		//DCタイムをゲット
		aPostprocessingDcTime[0]:=F_GetActualDcTime64();
	
		//1 コンテナ初期化
		hr := F_VN_CreateContainer(ipBoundingBoxes, ContainerType_Vector_TcVnRectangle_DINT, cNumBox, hr);		//NMS関数座標用
        hr := F_VN_CreateContainer(ipScores, ContainerType_Vector_REAL, cNumBox, hr);							//NMS関数スコア用
		
		hr := FW_SafeRelease(ADR(GVL.ipResultPoints));															//GVLにあるXY座標入力用コンテナをリリース(初回はコンテナ無いけど、大丈夫な関数)
		hr := F_VN_CreateContainer(GVL.ipResultPoints, ContainerType_Vector_TcVnPoint2_DINT, 0, hr);			//GVLにあるXY座標入力用コンテナ作成

		
		//2 Row Dataを座標用コンテナに書き込み
		nIteratorIdx:=0;		//インデックスリセット
		hr := F_VN_GetForwardIterator(ipBoundingBoxes, ipIterator, hr);		//座標用コンテナから前方走査イテレータを取得
		IF SUCCEEDED(hr) AND ipIterator <> 0 THEN
			hr := ipIterator.TcQueryInterface(IID_ITcVnAccess_TcVnRectangle_DINT, ADR(ipAccessTcVnRectangleDINT));		//TcVnRectangle_DINT型アクセス用のアクセスインターフェースをクエリ
			IF SUCCEEDED(hr) AND ipAccessTcVnRectangleDINT <> 0 THEN
				WHILE SUCCEEDED(hr) AND ipIterator.CheckIfEnd() <> S_OK DO		//コンテナの終端に達するまで高速ループ
					
					stRectangle.nX			:=REAL_TO_DINT(stModelOutput.out_output[0, nIteratorIdx, 0]-(stModelOutput.out_output[0, nIteratorIdx, 2]/2.0));		// 計算式： 左上X ＝ 中心X － (幅 ÷ 2)
					stRectangle.nY			:=REAL_TO_DINT(stModelOutput.out_output[0, nIteratorIdx, 1]-(stModelOutput.out_output[0, nIteratorIdx, 3]/2.0));		// 計算式： 左上Y ＝ 中心Y － (高さ ÷ 2)
					stRectangle.nWidth		:=REAL_TO_DINT(stModelOutput.out_output[0, nIteratorIdx, 2]);
					stRectangle.nHeight		:=REAL_TO_DINT(stModelOutput.out_output[0, nIteratorIdx, 3]);		//YOLOXセンター座標（cx, cy）から、TwinCAT左上座標（x, y）に変換して中間バッファのストラクトに書き込み
				
					hr := ipAccessTcVnRectangleDINT.Set(stRectangle);		//アクセスインターフェース経由でデータをコンテナに書き込み
					
					IF SUCCEEDED(hr) THEN
						hr := ipIterator.Increment();
						nIteratorIdx:=nIteratorIdx+1;
					END_IF
					
				END_WHILE
			END_IF
			hr := FW_SafeRelease(ADR(ipAccessTcVnRectangleDINT));		//アクセスインターフェースを解放
		END_IF 
		hr := FW_SafeRelease(ADR(ipIterator));		//イテレータを解放


		//3 Row Dataをスコア用コンテナに書き込み
		nIteratorIdx:=0;		//インデックスリセット
		hr := F_VN_GetForwardIterator(ipScores, ipIterator, hr);		//スコア用コンテナから前方走査イテレータを取得
		IF SUCCEEDED(hr) AND ipIterator <> 0 THEN
			hr := ipIterator.TcQueryInterface(IID_ITcVnAccess_REAL, ADR(ipAccessREAL));		//REAL型アクセス用のアクセスインターフェースをクエリ
			IF SUCCEEDED(hr) AND ipAccessREAL <> 0 THEN
				WHILE SUCCEEDED(hr) AND ipIterator.CheckIfEnd() <> S_OK DO		//コンテナの終端に達するまで高速ループ
					
					hr := ipAccessREAL.Set(stModelOutput.out_output[0, nIteratorIdx, 4] * stModelOutput.out_output[0, nIteratorIdx, 5]);		//アクセスインターフェース経由でデータをコンテナに書き込み
																																				//スコアはobj_score（物体らしさスコア）× class_score（クラススコア）					
					IF SUCCEEDED(hr) THEN
						hr := ipIterator.Increment();
						nIteratorIdx:=nIteratorIdx+1;
					END_IF
					
				END_WHILE
			END_IF
			hr := FW_SafeRelease(ADR(ipAccessREAL));		//アクセスインターフェースを解放
		END_IF 
		hr := FW_SafeRelease(ADR(ipIterator));		//イテレータを解放
		

		//4 Non-Maximum Suppression (NMS) の実行
        hr := F_VN_NonMaxSuppression(ipBoundingBoxes, ipScores, ipDestIndices, 0.3, 0.45, hr);		// 第4引数 (0.3)、第5引数（0.45）の説明コードの末尾にあり

		//NMS生存結果の抽出・描画・GVL出力
		hr := F_VN_GetNumberOfElements(ipDestIndices, nElementsFound, hr);		//NMSで生き残った（＝検出確定した）ワークの総数をカウント
		
		//1個以上ワークが検出された場合のみ、ループで1個ずつ処理を回す
		IF SUCCEEDED(hr) AND nElementsFound > 0 THEN
			
			FOR nIdx := 0 TO (ULINT_TO_UDINT(nElementsFound) - 1) DO
							
				hr := F_VN_GetAt_DINT(ipDestIndices, nTargetIndex, UDINT_TO_ULINT(nIdx), hr);		//NMSコンテナから、生き残った「元のRowDataのインデックス番号」を抽出

				hr := F_VN_GetAt_TcVnRectangle_DINT(ipBoundingBoxes, stFinalRect, DINT_TO_ULINT(nTargetIndex), hr);		//抽出したインデックスを使って、元の座標コンテナから長方形（Rect）データを取得
				
				hr := F_VN_GetAt_REAL(ipScores, fFinalScore, DINT_TO_ULINT(nTargetIndex), hr);		//抽出したインデックスを使って、元のスコアコンテナから確率データを取得

				// ONNXの座標から余白を引いて、縮小倍率で割り戻すことで、元画像のピクセル位置に戻す
				stFinalRect.nX      :=REAL_TO_DINT((DINT_TO_REAL(stFinalRect.nX) - fPadX) / fScale);
				stFinalRect.nY      :=REAL_TO_DINT((DINT_TO_REAL(stFinalRect.nY) - fPadY) / fScale);
				stFinalRect.nWidth  :=REAL_TO_DINT(DINT_TO_REAL(stFinalRect.nWidth) / fScale);
				stFinalRect.nHeight :=REAL_TO_DINT(DINT_TO_REAL(stFinalRect.nHeight) / fScale);
				
				//ワークの中心座標 (cx, cy) を計算し、DINT型構造体に落とし込む
				stCenterPoint[0]:=stFinalRect.nX + (stFinalRect.nWidth / 2);
				stCenterPoint[1]:=stFinalRect.nY + (stFinalRect.nHeight / 2);
				
				//確率表示にしたいので100倍
				fFinalScore:=fFinalScore*100.0;
				
				//ワーク幅から外れた物は無視
				IF (cWorkWidthMin<stFinalRect.nWidth AND stFinalRect.nWidth<cWorkWidthMax) AND (cWorkWidthMin<stFinalRect.nHeight AND stFinalRect.nHeight<cWorkWidthMax)  THEN
					
					//5 出力画像にワークの位置を画像に書き込み
					hr := F_VN_DrawRectangle(stFinalRect.nX, stFinalRect.nY, stFinalRect.nX+stFinalRect.nWidth, stFinalRect.nY + stFinalRect.nHeight,ipImageOut, aGreen, 2, hr);		//ワークを囲む長方形を描画
					
					hr := F_VN_DrawPoint(stCenterPoint[0], stCenterPoint[1], ipImageOut, TCVN_DS_PLUS, aGreen, hr);		//中心点に十字マークを描画
	
	
					//6 ワークのxy座標を画像に書き込み
					fbFormatString(	sFormat	:='( %2.1f ) = (%.3d, %.3d)', 
									arg1	:=F_REAL(fFinalScore),
									arg2	:=F_DINT(stCenterPoint[0]),
									arg3	:=F_DINT(stCenterPoint[1]));		//書き込み文字列生成
					
					hr := F_VN_PutText(fbFormatString.sOut, ipImageOut, stFinalRect.nX, stFinalRect.nY, TCVN_FT_HERSHEY_TRIPLEX, 0.5, aGreen, hr);		//XY座標を描画
					
					//7 GVLにあるコンテナにxy座標を書き込み
					hr := F_VN_AppendToContainer_TcVnVector2_DINT(stCenterPoint, GVL.ipResultPoints, hr);
				
				END_IF
				
			END_FOR
		END_IF
		
		//DCタイムをゲット
		aPostprocessingDcTime[1]:=F_GetActualDcTime64();
		
		iStep:=11;
		
	6..10:
		//NA

	11:
		//画面表示イメージを作成する
		hr := F_VN_TransformIntoDisplayableImage(ipImageIn, ipImageInDisp, hr);
        hr := F_VN_TransformIntoDisplayableImage(ipImageOut, ipImageOutDisp, hr);

		//ポインターの開放
		FW_SafeRelease(ADR(ipTensorImage));
		FW_SafeRelease(ADR(ipBoundingBoxes));
		FW_SafeRelease(ADR(ipScores));
		FW_SafeRelease(ADR(ipDestIndices));
		
		//各実行時間を計算[ms]
		lrPreprocessingTime		:=ULINT_TO_LREAL(aPreprocessingDcTime[1]-aPreprocessingDcTime[0]) / 1000000.0;
		lrInferenceTime			:=ULINT_TO_LREAL(aInferenceDcTime[1]-aInferenceDcTime[0]) / 1000000.0;
		lrPostprocessingTime	:=ULINT_TO_LREAL(aPostprocessingDcTime[1]-aPostprocessingDcTime[0]) / 1000000.0;
		
        iStep := 0;
		
	END_CASE







(*ワンポイントメモ

NMS処理の引数説明
0.3 ＝ スコアの閾値（足切りライン）正式な引数名はfScoreThreshold
意味：
*直前で計算した「obj_score × class_score」の最終スコアが、「0.3（30%）未満のゴミ候補は、重なりを調べる前に最初から全部切り捨てる」という設定です。
現場での調整イメージ：
*誤検出（ワークがないのに背景を誤認識する）が多いとき			:この値を 0.4 や 0.5 に上げます。より自信のある候補しか残らなくなります。
*見落とし（あるはずのワークをスルーしてしまう）が多いとき		:この値を 0.2 や 0.15 に下げます。少し自信がなくても候補として拾うようになります。

2. 0.45 ＝ 重複の閾値（ダブり判定の基準）正式な引数名は fOverlapThreshold
意味：
*1つのワークに対して、AIが何個もダブって四角枠（ボックス）を出してしまったときに、「面積の45%以上が重なっていたら、それは同じワークを二重検出しているとみなして、スコアが低い方を消す」という設定です。
※この重なりの割合をAIの世界では「IoU（Intersection over Union）」と呼びます。
現場での調整イメージ：
*1つのワークに四角枠が2個も3個も重なって残ってしまうとき								:この値を 0.3 や 0.35 に下げます（重なりの判定を厳しくして、ちょっとでも重なっていたら容赦なく1個にまとめます）。
*ワーク同士が実際に近くに密集していて、隣のワークの枠まで巻き添えで消されてしまうとき	:この値を 0.55 や 0.6 に上げます（かなりガッツリ重なっていない限り、別々のワークとして認めるようになります）。

*)

END_PROGRAM

// ---- 01_Submodules/Axis/FB_AxisVelocity.TcPOU
FUNCTION_BLOCK FB_AxisVelocity
VAR_OUTPUT
	// =============== State variables ========================
	bError			: BOOL;					// Error signal
	nErrorID		: UDINT;				// Error ID
	bMoves			: BOOL;					// Status of moving
END_VAR
VAR	
	// =============== Done signals of Halt and Reset =========
	bResetDone		: BOOL;					// Status of function block MC_Reset
	bHaltDone		: BOOL;					// Status of function block MC_Halt

	// =============== State variables ========================
	bStatusEnable	: BOOL;					// Enable feedback
	
	// =============== Velocity, override =====================
	fVelocity		: LREAL;				// Target velocity
	fOverride 		: LREAL := 100.0;		// Override 100%
	
	// =============== Trigger function blocks ================
	fbTriggerHalt	: R_TRIG;				// Trigger to recognize rising edge of halt input
	fbTriggerReset	: R_TRIG;				// Trigger to recognize rising edge of reset input
	
	// =============== Axis reference =========================
	AxisRef			: AXIS_REF;				// Axis reference (process data plc/nc)
	
	// =============== Motion function blocks =================
	fbMcPower 		: MC_Power;				// FB for enable and override
	fbMcReset 		: MC_Reset;				// FB to reset axis
	fbMcStop 		: MC_Stop;				// FB to stop axis
	fbMcHalt		: MC_Halt;				// FB to halt axis
	fbMcMove		: MC_MoveVelocity;		// FB to move axis (velocity movement)
END_VAR

// =========================================================
;
// =========================================================

PROPERTY bState_Enable : BOOL
GET
bState_Enable := bStatusEnable;
END_GET
END_PROPERTY

PROPERTY bState_HaltDone : BOOL
GET
bState_HaltDone := bHaltDone;
END_GET
END_PROPERTY

PROPERTY bState_ResetDone : BOOL
GET
bState_ResetDone := bResetDone;
END_GET
END_PROPERTY

METHOD Enable
VAR_INPUT
	bEnable		: BOOL;
END_VAR
// =========================================================

fbMCPower(	Enable 			:= bEnable, 
			Enable_Positive	:= bEnable, 
			Enable_Negative	:= bEnable, 
			Override		:= fOverride,
			Axis			:= AxisRef,
			Status			=> bStatusEnable);
			
IF fbMcPower.Error THEN
	bError		:= TRUE;
	nErrorID 	:= fbMcPower.ErrorID;
END_IF

AxisRef.ReadStatus();

bMoves := AxisRef.Status.Moving;

// =========================================================
END_METHOD

PROPERTY fTargetVelocity : LREAL
GET
fTargetVelocity := fVelocity;
END_GET
SET
fVelocity := fTargetVelocity;
END_SET
END_PROPERTY

METHOD Halt
VAR_INPUT
	bDriveHalt		: BOOL;					// Request stop
END_VAR
// =========================================================

IF bDriveHalt THEN
	// Move Execute FALSE
	fbMCMove(	Execute	:= FALSE,
				Axis 	:= AxisRef);
ELSE
	// Reset done signal
	bHaltDone := FALSE;
END_IF

// Trigger
fbTriggerHalt(CLK := bDriveHalt);

IF fbTriggerHalt.Q THEN
	fbMcHalt(	Execute	:= TRUE,
				Axis 	:= AxisRef);
ELSE
	fbMcHalt(Axis := AxisRef);
END_IF

// Done / Error / Command aborted
IF fbMcHalt.Done OR fbMcHalt.Error OR fbMcHalt.CommandAborted THEN
	bError		:= fbMcHalt.Error;
	nErrorID 	:= fbMcHalt.ErrorID;
	bHaltDone 	:= fbMcHalt.Done;
	
	fbMCMove(	Execute	:= FALSE,
				Axis 	:= AxisRef);
				
	fbMcHalt(	Execute	:= FALSE,
				Axis 	:= AxisRef);
END_IF

// =========================================================
END_METHOD

METHOD MoveBw
VAR_INPUT
END_VAR
// =========================================================

// Not error
IF NOT fbMcMove.Error THEN
	fbMCMove(	Execute 	:= TRUE,
				Velocity 	:= fVelocity,
				Direction 	:= MC_Negative_Direction,
				Axis 		:= AxisRef );
END_IF

// Error / Command aborted
IF fbMCMove.Error OR fbMCMove.CommandAborted THEN
	IF fbMcMove.Error THEN
		bError		:= TRUE;
		nErrorID 	:= fbMCMove.ErrorID;
	END_IF
	
	fbMCMove(	Execute	:= FALSE,
				Axis 	:= AxisRef);
END_IF

// =========================================================
END_METHOD

METHOD MoveFw
VAR_INPUT
END_VAR
// =========================================================

// Not error
IF NOT fbMcMove.Error THEN
	fbMCMove(	Execute 	:= TRUE,
				Velocity 	:= fVelocity,
				Direction 	:= MC_Positive_Direction,
				Axis 		:= AxisRef );
END_IF

// Error / Command aborted
IF fbMCMove.Error OR fbMCMove.CommandAborted THEN
	IF fbMcMove.Error THEN
		bError		:= TRUE;
		nErrorID 	:= fbMCMove.ErrorID;
	END_IF
	
	fbMCMove(	Execute	:= FALSE,
				Axis 	:= AxisRef);
END_IF

// =========================================================
END_METHOD

METHOD Reset
VAR_INPUT
	bDriveReset		: BOOL;					// Request reset
END_VAR
// =========================================================

IF NOT bDriveReset THEN
	bResetDone 	:= FALSE;
END_IF

// Trigger
fbTriggerReset(CLK := bDriveReset);

IF fbTriggerReset.Q THEN
	bHaltDone 	:= FALSE;
	
	fbMcReset(Execute := TRUE, Axis := AxisRef);
ELSE
	fbMcReset(Axis := AxisRef);
END_IF

// Done / Error
IF fbMcReset.Done OR fbMcReset.Error THEN
	bError		:= fbMcReset.Error;
	nErrorID 	:= fbMcReset.ErrorID;
	bResetDone 	:= fbMcReset.Done;

	fbMcReset(	Execute	:= FALSE,
				Axis 	:= AxisRef);
END_IF

// =========================================================
END_METHOD

METHOD Stop
VAR_INPUT
	bDriveStop		: BOOL;					// Request stop
END_VAR
// =========================================================

IF bDriveStop THEN
	// Move Execute FALSE
	fbMCMove(	Execute	:= FALSE,
				Axis 	:= AxisRef);
ELSE
	// Reset done signal
	bHaltDone := FALSE;
END_IF

// Trigger
fbTriggerHalt(CLK := bDriveStop);

IF fbTriggerHalt.Q THEN
	fbMcStop(	Execute	:= TRUE,
				Axis 	:= AxisRef);
ELSE
	fbMcStop(Axis := AxisRef);
END_IF

// Done / Error / Command aborted
IF fbMcStop.Done OR fbMcStop.Error OR fbMcStop.CommandAborted THEN
	bError		:= fbMcStop.Error;
	nErrorID 	:= fbMcStop.ErrorID;
	bHaltDone 	:= fbMcStop.Done;
	
	fbMCMove(	Execute	:= FALSE,
				Axis 	:= AxisRef);
				
	fbMcStop(	Execute	:= FALSE,
				Axis 	:= AxisRef);
END_IF

// =========================================================
END_METHOD

END_FUNCTION_BLOCK

// ---- 01_Submodules/LoadCell/RowLoadCell/FB_LoadCell_ForRowValue.TcPOU
FUNCTION_BLOCK FB_LoadCell_ForRowValue
VAR_INPUT
	diBridgeInputs			AT %I*	:DINT;			//ロードセルの出力電圧生値
	diSupplyInputs			AT %I*	:DINT;			//ロードセルへの印加電圧生値
	
END_VAR
VAR_OUTPUT
END_VAR
VAR PERSISTENT
	_lrTareWeight					:LREAL;			//風袋重量[kg]
END_VAR
VAR
	_lrCalibrationWeight			:LREAL;			//校正重量[kg]		

	_lrBridgeVoltage				:LREAL;			//ロードセルの出力電圧[mV]
	_lrSupplyVoltage				:LREAL;			//ロードセルへの印加電圧[V]
	_lrGrossWeight					:LREAL;			//測定重量[kg]
	_lrNetWeight					:LREAL;			//正味重量[kg]
	
	lrSlope							:LREAL;			//校正後の傾き
	
	lrRatedCapacity					:LREAL;			//ロードセル定格容量　R.C. [kg]
	lrRatedOutput					:LREAL;			//ロードセル定格出力 R.O. [mV/V]
	
	diMaxNumber						:DINT;			//ロードセル入力ターミナル最大値　
	diBridgeMeasuringRange			:DINT;			//ロードセルの出力電圧入力ターミナル測定レンジ　[mV]
	lrSupplyMeasuringRange			:LREAL;			//ロードセルへの印加電圧入力ターミナル測定レンジ [V]
END_VAR

METHOD CalibrationWeightSet
VAR_INPUT
	bCalibrationWeightSet	:BOOL;
END_VAR
VAR
	lrNowGrossWeight		:LREAL;
END_VAR
	IF bCalibrationWeightSet=TRUE THEN
		
		//今のグロスウェイト確認[kg]
		IF diSupplyInputs<>0 AND diBridgeMeasuringRange<>0  AND lrRatedOutput<>0 THEN
			lrNowGrossWeight:=((DINT_TO_LREAL(diBridgeInputs)*DINT_TO_LREAL(diBridgeMeasuringRange))/(DINT_TO_LREAL(diSupplyInputs)*lrSupplyMeasuringRange))*(lrRatedCapacity/lrRatedOutput);
		END_IF
		
		//今のグロスウェイトが風袋重量より重いことを確認
		IF _lrTareWeight+0.010 < lrNowGrossWeight THEN
			//切片を計算
			IF lrNowGrossWeight<>0 AND _lrTareWeight<>0 THEN
				lrSlope:=(_lrCalibrationWeight-0)/(lrNowGrossWeight-_lrTareWeight);
			END_IF
		END_IF
		
	END_IF
END_METHOD

//FB_Init は常に暗黙的に使用可能で、主に初期化に使用されます。
//戻り値は評価されません。特定の結果を得るために、メソッドを明示的に宣言し、
//そのメソッドに標準の初期化コードをもったコードを追加することができます。戻り値を評価できます。
METHOD FB_Init: BOOL
VAR_INPUT
    bInitRetains: BOOL; // TRUE: 保持変数は初期化されます (ウォーム リセット、あるいはコールド リセット)
    bInCopyCode: BOOL;  // TRUE: 後でコードをコピーする (オンライン変更) ために、インスタンスをコピーします。
		
	lrRatedCapacity				:LREAL;			//ロードセル定格容量　R.C. [kg]
	lrRatedOutput				:LREAL;			//ロードセル定格出力 R.O. [mV/V]
	
	diMaxNumber					:DINT;			//ロードセル入力ターミナル最大値　
	diBridgeMeasuringRange		:DINT;			//ロードセルの出力電圧入力ターミナル測定レンジ　[mV]
	lrSupplyMeasuringRange		:LREAL;			//ロードセルへの印加電圧入力ターミナル測定レンジ [V]
END_VAR
THIS^.lrRatedCapacity			:=lrRatedCapacity;
THIS^.lrRatedOutput				:=lrRatedOutput;

THIS^.diMaxNumber				:=diMaxNumber;
THIS^.diBridgeMeasuringRange	:=diBridgeMeasuringRange;
THIS^.lrSupplyMeasuringRange	:=lrSupplyMeasuringRange;
END_METHOD

PROPERTY lrBridgeVoltage : LREAL
GET
	//ロードセルの出力電圧計算[mV]
	IF diMaxNumber<>0 THEN
		_lrBridgeVoltage:=DINT_TO_LREAL(diBridgeInputs)*(DINT_TO_LREAL(diBridgeMeasuringRange)/diMaxNumber);
	END_IF
	
	lrBridgeVoltage:=_lrBridgeVoltage;
END_GET
END_PROPERTY

PROPERTY lrCalibrationWeight : LREAL
SET
_lrCalibrationWeight:=lrCalibrationWeight;
END_SET
END_PROPERTY

PROPERTY lrGrossWeight : LREAL
GET
	//グロスウェイト計算[kg]
	IF diSupplyInputs<>0 and diBridgeMeasuringRange<>0  AND lrRatedOutput<>0 THEN
		_lrGrossWeight:=((DINT_TO_LREAL(diBridgeInputs)*DINT_TO_LREAL(diBridgeMeasuringRange))/(DINT_TO_LREAL(diSupplyInputs)*lrSupplyMeasuringRange))*(lrRatedCapacity/lrRatedOutput);
	END_IF
	
	lrGrossWeight:=_lrGrossWeight;
END_GET
END_PROPERTY

PROPERTY lrNetWeight : LREAL
GET
	//ネットウェイト計算[kg]
	_lrNetWeight:=_lrGrossWeight-_lrTareWeight;
	
	lrNetWeight:=_lrNetWeight;
END_GET
END_PROPERTY

PROPERTY lrSupplyVoltage : LREAL
GET
	//ロードセルへの印加電圧計算[V]
	IF diMaxNumber<>0 THEN
		_lrSupplyVoltage:=DINT_TO_LREAL(diSupplyInputs)*(lrSupplyMeasuringRange/diMaxNumber);
	END_IF
	
	lrSupplyVoltage:=_lrSupplyVoltage;
END_GET
END_PROPERTY

PROPERTY lrTareWeight : LREAL
GET
lrTareWeight:=_lrTareWeight;
END_GET
END_PROPERTY

METHOD TareWeightSet
VAR_INPUT
	bTareWeightSet					:BOOL;
	bPersistentDataWriteRequest		:REFERENCE TO BOOL;
END_VAR
	//風袋重量セット[kg]	
	IF bTareWeightSet=TRUE THEN
		
		IF diSupplyInputs<>0 AND diBridgeMeasuringRange<>0  AND lrRatedOutput<>0 THEN
			_lrTareWeight:=((DINT_TO_LREAL(diBridgeInputs)*DINT_TO_LREAL(diBridgeMeasuringRange))/(DINT_TO_LREAL(diSupplyInputs)*lrSupplyMeasuringRange))*(lrRatedCapacity/lrRatedOutput);
			
			bPersistentDataWriteRequest:=TRUE;
			
		END_IF
		
	ELSE
		bPersistentDataWriteRequest:=FALSE;
	END_IF
END_METHOD

END_FUNCTION_BLOCK

// ---- 01_Submodules/PcManagement/1sUPS/FB_1sUPS_CX81xx.TcPOU
FUNCTION_BLOCK FB_1sUPS_CX81xx IMPLEMENTS i1sUPS
VAR
	fb1sUps		:FB_S_UPS_CX81xx;
END_VAR

PROPERTY bPowerFailDetect : BOOL
GET
bPowerFailDetect:=fb1sUps.bPowerFailDetect;
END_GET
END_PROPERTY

PROPERTY eUpsState : E_S_UPS_State
GET
eUpsState := fb1sUps.eState;
END_GET
END_PROPERTY

METHOD UPSCall
VAR_INPUT
	(*PC AMS Net ID*)
	PcAmsNetId	: AMSNETID;
END_VAR
fb1sUps(sNetID				:=F_CreateAmsNetId(PcAmsNetId),
		iPLCPort			:=_AppInfo.AdsPort,
		tTimeout			:=DEFAULT_ADS_TIMEOUT,
		eUpsMode			:=E_S_UPS_Mode.eSUPS_WrPersistData_Shutdown,
		ePersistentMode		:=E_PersistentMode.SPDM_2PASS,
		tRecoverTime		:=T#10S,
		bPowerFailDetect	=>,
		eState				=>
		);
END_METHOD

END_FUNCTION_BLOCK

// ---- 04_Application/Vision/FB_Pixel_TO_Coordinate.TcPOU
FUNCTION_BLOCK FB_Pixel_TO_Coordinate
VAR_INPUT
	lrUPixel		:LREAL;		// 入力: 画像座標 [px]
	lrVPixel		:LREAL;		// 入力: 画像座標 [px]
END_VAR
VAR_OUTPUT
	lrXCoordinate	:LREAL;		// 出力: 盤面座標 [mm]
	lrYCoordinate	:LREAL;		// 出力: 盤面座標 [mm]
	
	bError			:bool;		// エラー
END_VAR
VAR
	xh				:LREAL;		// 計算用中間変数
	yh				:LREAL;		// 計算用中間変数
	wh				:LREAL;		// 計算用中間変数
    
    // 1行目:X係数, 2行目:Y係数, 3行目:分母係数
    H				:ARRAY[1..3, 1..3] OF LREAL:=	[
													0.4956,  -0.0012,  -56.4406,	// h11, h12, h13 (1行目)
													-0.0038,   0.4965,   -7.3795,	// h21, h22, h23 (2行目)
													0.0000,   0.0000,    1.0000		// h31, h32, h33 (3行目)
													];
END_VAR

// Xの分子: h11*u + h12*v + h13
xh := lrUPixel * H[1,1] + lrVPixel * H[1,2] + H[1,3];

// Yの分子: h21*u + h22*v + h23
yh := lrUPixel * H[2,1] + lrVPixel * H[2,2] + H[2,3];

// 分母 (Weight): h31*u + h32*v + h33
wh := lrUPixel * H[3,1] + lrVPixel * H[3,2] + H[3,3];


// ゼロ割り算の防止と実座標への変換
IF wh <> 0.0 THEN
    lrXCoordinate := xh / wh;
    lrYCoordinate := yh / wh;
	
	bError:=FALSE;
ELSE
    lrXCoordinate := 0.0;
    lrYCoordinate := 0.0;
	
	bError:=TRUE;
END_IF

END_FUNCTION_BLOCK

// ---- POUs/FB_MotionShapeWrite.TcPOU
FUNCTION_BLOCK FB_MotionShapeWrite
VAR
	bStart				:BOOL;
	bEnd				:BOOL;
	
	pMcMoveAbs			:ARRAY[E_Axis.X_Axis..E_Axis.Gripper] OF POINTER TO MC_MoveAbsolute;
	pMcMoveAbsSub		:ARRAY[E_Axis.X_Axis..E_Axis.Z_Axis] OF POINTER TO MC_MoveAbsolute;
	
	i					:INT;
	iNext				:INT:=0;
	eStep				:E_CircleEllipseWriteStep:=E_CircleEllipseWriteStep.Check;
	iStep				:INT:=0;
	lrDeg				:LREAL :=0;

	fbZAxisTPCon0		:FB_Z_Axis_TargetPositionConvert;
	fbZAxisTPCon1		:FB_Z_Axis_TargetPositionConvert;
	bCheck0				:ARRAY[E_Axis.X_Axis..E_Axis.Z_Axis] OF BOOL;
	bCheck1				:ARRAY[E_Axis.X_Axis..E_Axis.Z_Axis] OF BOOL;
	
	//円用の変数
	iEndNumberCircle	:INT;(*書き終わった円の個数*)
	iWrittingCircle		:INT;(*今から何個目の円を書くのか*)
	stCircleSettings	:ARRAY[1..32] OF ST_CircleSettings;
	
	//楕円用の変数
	iEndNumberEllipse	:INT;(*書き終わった楕円の個数*)
	iWrittingEllipse	:INT;(*今から何個目の楕円を書くのか*)
	stEllipseSettings	:ARRAY[1..32] OF ST_EllipseSetting;
	lrBase0				:ARRAY[E_Axis.X_Axis..E_Axis.Y_Axis] OF LREAL;
	lrBase1				:ARRAY[E_Axis.X_Axis..E_Axis.Y_Axis] OF LREAL;
END_VAR

IF bStart<>TRUE THEN
	RETURN;
END_IF

CASE iNext OF
	0:
		eStep:=E_CircleEllipseWriteStep.Check;
		iStep:=0;
		i:=0;
		iEndNumberCircle:=0;
		iWrittingCircle:=0;
		iEndNumberEllipse:=0;
		iWrittingEllipse:=0;
		iNext:=2;

	2:
		CircleMeth();
	
	3:
		EllipseMeth();
	
	4:
		bEnd:=TRUE;
		iNext:=0;
		
END_CASE

PROPERTY bEndProp : BOOL
GET
bEndprop:=bEnd;
END_GET
SET
bEnd:=bEndProp;
END_SET
END_PROPERTY

PROPERTY bStartProp : BOOL
GET
bStartprop:=bStart;
END_GET
SET
bStart:=bStartProp;
END_SET
END_PROPERTY

METHOD CircleMeth : BOOL
VAR_INPUT
END_VAR
CASE eStep OF

E_CircleEllipseWriteStep.Check:(*まず書く円を確認*)

	iEndNumberCircle:=iWrittingCircle;
	iWrittingCircle:=0;

	FOR i :=  iEndNumberCircle + 1 TO 32 BY 1 DO
		IF stCircleSettings[i].bWrite=TRUE THEN
			iWrittingCircle:=i;
			eStep:=E_CircleEllipseWriteStep.FirstPotisionMove;
			EXIT;
		END_IF
	END_FOR

	IF iWrittingCircle=0 THEN
		iNext:=3;
	END_IF

E_CircleEllipseWriteStep.FirstPotisionMove:(*円の書き始め位置へ移動*)

	CASE iStep OF
	0:
		iStep:=1;
		lrDeg:=stCircleSettings[iWrittingCircle].lrStartDeg;
		
	1:
		pMcMoveAbs[E_Axis.X_Axis]^.Execute:=TRUE;
		pMcMoveAbs[E_Axis.Y_Axis]^.Execute:=TRUE;
		pMcMoveAbs[E_Axis.X_Axis]^.Position:=stCircleSettings[iWrittingCircle].uiXCenter + stCircleSettings[iWrittingCircle].uiRadius * COS(lrDeg*PI/180);
		pMcMoveAbs[E_Axis.Y_Axis]^.Position:=stCircleSettings[iWrittingCircle].uiYCenter + stCircleSettings[iWrittingCircle].uiRadius * SIN(lrDeg*PI/180);
		pMcMoveAbs[E_Axis.X_Axis]^.Velocity:=150;
		pMcMoveAbs[E_Axis.Y_Axis]^.Velocity:=150;

		IF pMcMoveAbs[E_Axis.X_Axis]^.Done=TRUE AND pMcMoveAbs[E_Axis.Y_Axis]^.Done=TRUE THEN
			iStep:=2;
			pMcMoveAbs[E_Axis.X_Axis]^.Execute:=FALSE;
			pMcMoveAbs[E_Axis.Y_Axis]^.Execute:=FALSE;
		END_IF;
		
	2:
		pMcMoveAbs[E_Axis.Z_Axis]^.Execute:=TRUE;
		pMcMoveAbs[E_Axis.Z_Axis]^.Velocity:=150;
		
		fbZAxisTPCon0(
			lrX_AxisTP		:=pMcMoveAbs[E_Axis.X_Axis]^.Position,
			lrY_AxisTP		:=pMcMoveAbs[E_Axis.Y_Axis]^.Position,
			lrZ_AxisTP		:=273-GVL.lrPenFullLength+GVL.lrPenGripLength,
			lrZ_AxisConTP	=>pMcMoveAbs[E_Axis.Z_Axis]^.Position
			);
				
		IF pMcMoveAbs[E_Axis.Z_Axis]^.Done=TRUE THEN
			eStep:=E_CircleEllipseWriteStep.Write;
			pMcMoveAbs[E_Axis.Z_Axis]^.Execute:=FALSE;
			iStep:=0;
		END_IF;
	
	END_CASE;

E_CircleEllipseWriteStep.Write:(*円を書いていく*)

	CASE iStep OF
	0:
		bCheck0[E_Axis.X_Axis]:=TRUE;
		bCheck1[E_Axis.X_Axis]:=TRUE;
		bCheck0[E_Axis.Y_Axis]:=TRUE;
		bCheck1[E_Axis.Y_Axis]:=TRUE;
		bCheck0[E_Axis.Z_Axis]:=TRUE;
		bCheck1[E_Axis.Z_Axis]:=TRUE;
		lrDeg:=stCircleSettings[iWrittingCircle].lrStartDeg;
		iStep:=1;

	1:	
		IF pMcMoveAbs[E_Axis.X_Axis]^.Done=TRUE THEN bCheck0[E_Axis.X_Axis]:=TRUE; END_IF;
		IF pMcMoveAbsSub[E_Axis.X_Axis]^.Done=TRUE THEN bCheck1[E_Axis.X_Axis]:=TRUE; END_IF;
		IF pMcMoveAbs[E_Axis.Y_Axis]^.Done=TRUE THEN bCheck0[E_Axis.Y_Axis]:=TRUE; END_IF;
		IF pMcMoveAbsSub[E_Axis.Y_Axis]^.Done=TRUE THEN bCheck1[E_Axis.Y_Axis]:=TRUE; END_IF;
		IF pMcMoveAbs[E_Axis.Z_Axis]^.Done=TRUE THEN bCheck0[E_Axis.Z_Axis]:=TRUE; END_IF;
		IF pMcMoveAbsSub[E_Axis.Z_Axis]^.Done=TRUE THEN bCheck1[E_Axis.Z_Axis]:=TRUE; END_IF;
	
		IF bCheck0[E_Axis.X_Axis]=TRUE AND bCheck0[E_Axis.Y_Axis]=TRUE AND bCheck0[E_Axis.Z_Axis]=TRUE THEN
			bCheck0[E_Axis.X_Axis]:=FALSE;	
			bCheck0[E_Axis.Y_Axis]:=FALSE;
			bCheck0[E_Axis.Z_Axis]:=FALSE;
			lrDeg:=lrDeg + 1;
			pMcMoveAbs[E_Axis.X_Axis]^.Position:=stCircleSettings[iWrittingCircle].uiXCenter + stCircleSettings[iWrittingCircle].uiRadius * COS(lrDeg*PI/180);
			pMcMoveAbs[E_Axis.Y_Axis]^.Position:=stCircleSettings[iWrittingCircle].uiYCenter + stCircleSettings[iWrittingCircle].uiRadius * SIN(lrDeg*PI/180);
			
			fbZAxisTPCon0(
				lrX_AxisTP		:=pMcMoveAbs[E_Axis.X_Axis]^.Position,
				lrY_AxisTP		:=pMcMoveAbs[E_Axis.Y_Axis]^.Position,
				lrZ_AxisTP		:=273-GVL.lrPenFullLength+GVL.lrPenGripLength,
				lrZ_AxisConTP	=>pMcMoveAbs[E_Axis.Z_Axis]^.Position
				);

			pMcMoveAbs[E_Axis.X_Axis]^.Execute:=TRUE;
			pMcMoveAbs[E_Axis.Y_Axis]^.Execute:=TRUE;
			pMcMoveAbs[E_Axis.Z_Axis]^.Execute:=TRUE;
			pMcMoveAbs[E_Axis.X_Axis]^.Velocity:=150;
			pMcMoveAbs[E_Axis.Y_Axis]^.Velocity:=150;
			pMcMoveAbs[E_Axis.Z_Axis]^.Velocity:=150;
		ELSE
			pMcMoveAbs[E_Axis.X_Axis]^.Execute:=FALSE;
			pMcMoveAbs[E_Axis.Y_Axis]^.Execute:=FALSE;
			pMcMoveAbs[E_Axis.Z_Axis]^.Execute:=FALSE;
		END_IF;
		
		IF bCheck1[E_Axis.X_Axis]=TRUE AND bCheck1[E_Axis.Y_Axis]=TRUE AND bCheck1[E_Axis.Z_Axis]=TRUE THEN
			bCheck1[E_Axis.X_Axis]:=FALSE;	
			bCheck1[E_Axis.Y_Axis]:=FALSE;
			bCheck1[E_Axis.Z_Axis]:=FALSE;
			lrDeg:=lrDeg + 1;
			pMcMoveAbsSub[E_Axis.X_Axis]^.Position:=stCircleSettings[iWrittingCircle].uiXCenter + stCircleSettings[iWrittingCircle].uiRadius * COS(lrDeg*PI/180);
			pMcMoveAbsSub[E_Axis.Y_Axis]^.Position:=stCircleSettings[iWrittingCircle].uiYCenter + stCircleSettings[iWrittingCircle].uiRadius * SIN(lrDeg*PI/180);
			
			fbZAxisTPCon1(
				lrX_AxisTP		:=pMcMoveAbsSub[E_Axis.X_Axis]^.Position,
				lrY_AxisTP		:=pMcMoveAbsSub[E_Axis.Y_Axis]^.Position,
				lrZ_AxisTP		:=273-GVL.lrPenFullLength+GVL.lrPenGripLength,
				lrZ_AxisConTP	=>pMcMoveAbsSub[E_Axis.Z_Axis]^.Position
				);

			pMcMoveAbsSub[E_Axis.X_Axis]^.Execute:=TRUE;
			pMcMoveAbsSub[E_Axis.Y_Axis]^.Execute:=TRUE;
			pMcMoveAbsSub[E_Axis.Z_Axis]^.Execute:=TRUE;
			pMcMoveAbsSub[E_Axis.X_Axis]^.Velocity:=150;
			pMcMoveAbsSub[E_Axis.Y_Axis]^.Velocity:=150;
			pMcMoveAbsSub[E_Axis.Z_Axis]^.Velocity:=150;
		ELSE
			pMcMoveAbsSub[E_Axis.X_Axis]^.Execute:=FALSE;
			pMcMoveAbsSub[E_Axis.Y_Axis]^.Execute:=FALSE;
			pMcMoveAbsSub[E_Axis.Z_Axis]^.Execute:=FALSE;
		END_IF;
	
		IF stCircleSettings[iWrittingCircle].lrEndDeg < lrDeg THEN
			pMcMoveAbs[E_Axis.X_Axis]^.Execute:=FALSE;
			pMcMoveAbs[E_Axis.Y_Axis]^.Execute:=FALSE;
			pMcMoveAbs[E_Axis.Z_Axis]^.Execute:=FALSE;
			pMcMoveAbsSub[E_Axis.X_Axis]^.Execute:=FALSE;
			pMcMoveAbsSub[E_Axis.Y_Axis]^.Execute:=FALSE;
			pMcMoveAbsSub[E_Axis.Z_Axis]^.Execute:=FALSE;
			eStep:=E_CircleEllipseWriteStep.ZAxisUpPotision;
			iStep:=0;
			lrDeg:=0;
		END_IF;
	
	END_CASE;

E_CircleEllipseWriteStep.ZAxisUpPotision:(*Z軸を持ち上げる、ペンが紙に当たらないように*)

	pMcMoveAbs[E_Axis.Z_Axis]^.Execute:=TRUE;
	pMcMoveAbs[E_Axis.Z_Axis]^.Position:=273-GVL.lrPenFullLength+GVL.lrPenGripLength-50;
	pMcMoveAbs[E_Axis.Z_Axis]^.Velocity:=150;

	IF pMcMoveAbs[E_Axis.Z_Axis]^.Done=TRUE THEN
		eStep:=E_CircleEllipseWriteStep.Check;
		pMcMoveAbs[E_Axis.Z_Axis]^.Execute:=FALSE;
	END_IF;
	
END_CASE;
END_METHOD

METHOD EllipseMeth : BOOL
VAR_INPUT
END_VAR
CASE eStep OF
	
E_CircleEllipseWriteStep.Check:(*まず書く楕円を確認*)
	
	iEndNumberEllipse:=iWrittingEllipse;
	iWrittingEllipse:=0;

	FOR i :=  iEndNumberEllipse + 1 TO 32 BY 1 DO
		IF stEllipseSettings[i].bWrite=TRUE THEN
			iWrittingEllipse:=i;
			eStep:=E_CircleEllipseWriteStep.FirstPotisionMove;
			EXIT;
		END_IF
	END_FOR

	IF iWrittingEllipse=0 THEN
		iNext:=4;
	END_IF
	
E_CircleEllipseWriteStep.FirstPotisionMove:(*楕円の書き始め位置へ移動*)
	
	CASE iStep OF
	0:
		iStep:=1;
		lrDeg:=stEllipseSettings[iWrittingEllipse].lrStartDeg;
	
	1:
		lrBase0[E_Axis.X_Axis]:= stEllipseSettings[iWrittingEllipse].uiVertex * COS(lrDeg*PI/180);
		lrBase0[E_Axis.Y_Axis]:= stEllipseSettings[iWrittingEllipse].uiCoVertex * SIN(lrDeg*PI/180);
		pMcMoveAbs[E_Axis.X_Axis]^.Execute:=TRUE;
		pMcMoveAbs[E_Axis.Y_Axis]^.Execute:=TRUE;
		pMcMoveAbs[E_Axis.X_Axis]^.Position:=stEllipseSettings[iWrittingEllipse].uiXCenter + lrBase0[E_Axis.X_Axis] * COS(stEllipseSettings[iWrittingEllipse].lrSlopeDeg*PI/180) - lrBase0[E_Axis.Y_Axis] * SIN(stEllipseSettings[iWrittingEllipse].lrSlopeDeg*PI/180);
		pMcMoveAbs[E_Axis.Y_Axis]^.Position:=stEllipseSettings[iWrittingEllipse].uiYCenter + lrBase0[E_Axis.X_Axis] * SIN(stEllipseSettings[iWrittingEllipse].lrSlopeDeg*PI/180) + lrBase0[E_Axis.Y_Axis] * COS(stEllipseSettings[iWrittingEllipse].lrSlopeDeg*PI/180);
		pMcMoveAbs[E_Axis.X_Axis]^.Velocity:=150;
		pMcMoveAbs[E_Axis.Y_Axis]^.Velocity:=150;

		IF pMcMoveAbs[E_Axis.X_Axis]^.Done=TRUE AND pMcMoveAbs[E_Axis.Y_Axis]^.Done=TRUE THEN
			iStep:=2;
			pMcMoveAbs[E_Axis.X_Axis]^.Execute:=FALSE;
			pMcMoveAbs[E_Axis.Y_Axis]^.Execute:=FALSE;
		END_IF;
		
	2:
		pMcMoveAbs[E_Axis.Z_Axis]^.Execute:=TRUE;
		pMcMoveAbs[E_Axis.Z_Axis]^.Velocity:=150;
		
		fbZAxisTPCon0(
			lrX_AxisTP		:=pMcMoveAbs[E_Axis.X_Axis]^.Position,
			lrY_AxisTP		:=pMcMoveAbs[E_Axis.Y_Axis]^.Position,
			lrZ_AxisTP		:=273-GVL.lrPenFullLength+GVL.lrPenGripLength,
			lrZ_AxisConTP	=>pMcMoveAbs[E_Axis.Z_Axis]^.Position
			);
				
		IF pMcMoveAbs[E_Axis.Z_Axis]^.Done=TRUE THEN
			eStep:=E_CircleEllipseWriteStep.Write;
			pMcMoveAbs[E_Axis.Z_Axis]^.Execute:=FALSE;
			iStep:=0;
		END_IF;
		
	END_CASE
	
E_CircleEllipseWriteStep.Write:(*楕円を書いていく*)

	CASE iStep OF
	0:
		bCheck0[E_Axis.X_Axis]:=TRUE;
		bCheck1[E_Axis.X_Axis]:=TRUE;
		bCheck0[E_Axis.Y_Axis]:=TRUE;
		bCheck1[E_Axis.Y_Axis]:=TRUE;
		bCheck0[E_Axis.Z_Axis]:=TRUE;
		bCheck1[E_Axis.Z_Axis]:=TRUE;
		lrDeg:=stEllipseSettings[iWrittingEllipse].lrStartDeg;
		iStep:=1;

	1:	
		IF pMcMoveAbs[E_Axis.X_Axis]^.Done=TRUE THEN bCheck0[E_Axis.X_Axis]:=TRUE; END_IF;
		IF pMcMoveAbsSub[E_Axis.X_Axis]^.Done=TRUE THEN bCheck1[E_Axis.X_Axis]:=TRUE; END_IF;
		IF pMcMoveAbs[E_Axis.Y_Axis]^.Done=TRUE THEN bCheck0[E_Axis.Y_Axis]:=TRUE; END_IF;
		IF pMcMoveAbsSub[E_Axis.Y_Axis]^.Done=TRUE THEN bCheck1[E_Axis.Y_Axis]:=TRUE; END_IF;
		IF pMcMoveAbs[E_Axis.Z_Axis]^.Done=TRUE THEN bCheck0[E_Axis.Z_Axis]:=TRUE; END_IF;
		IF pMcMoveAbsSub[E_Axis.Z_Axis]^.Done=TRUE THEN bCheck1[E_Axis.Z_Axis]:=TRUE; END_IF;

		IF bCheck0[E_Axis.X_Axis]=TRUE AND bCheck0[E_Axis.Y_Axis]=TRUE AND bCheck0[E_Axis.Z_Axis]=TRUE THEN
			bCheck0[E_Axis.X_Axis]:=FALSE;	
			bCheck0[E_Axis.Y_Axis]:=FALSE;
			bCheck0[E_Axis.Z_Axis]:=FALSE;
			lrDeg:=lrDeg + 1;
			lrBase0[E_Axis.X_Axis]:= stEllipseSettings[iWrittingEllipse].uiVertex * COS(lrDeg*PI/180);
			lrBase0[E_Axis.Y_Axis]:= stEllipseSettings[iWrittingEllipse].uiCoVertex * SIN(lrDeg*PI/180);
			pMcMoveAbs[E_Axis.X_Axis]^.Position:=stEllipseSettings[iWrittingEllipse].uiXCenter + lrBase0[E_Axis.X_Axis] * COS(stEllipseSettings[iWrittingEllipse].lrSlopeDeg*PI/180) - lrBase0[E_Axis.Y_Axis] * SIN(stEllipseSettings[iWrittingEllipse].lrSlopeDeg*PI/180);
			pMcMoveAbs[E_Axis.Y_Axis]^.Position:=stEllipseSettings[iWrittingEllipse].uiYCenter + lrBase0[E_Axis.X_Axis] * SIN(stEllipseSettings[iWrittingEllipse].lrSlopeDeg*PI/180) + lrBase0[E_Axis.Y_Axis] * COS(stEllipseSettings[iWrittingEllipse].lrSlopeDeg*PI/180);
			
			fbZAxisTPCon0(
				lrX_AxisTP		:=pMcMoveAbs[E_Axis.X_Axis]^.Position,
				lrY_AxisTP		:=pMcMoveAbs[E_Axis.Y_Axis]^.Position,
				lrZ_AxisTP		:=273-GVL.lrPenFullLength+GVL.lrPenGripLength,
				lrZ_AxisConTP	=>pMcMoveAbs[E_Axis.Z_Axis]^.Position
				);

			pMcMoveAbs[E_Axis.X_Axis]^.Execute:=TRUE;
			pMcMoveAbs[E_Axis.Y_Axis]^.Execute:=TRUE;
			pMcMoveAbs[E_Axis.Z_Axis]^.Execute:=TRUE;
			pMcMoveAbs[E_Axis.X_Axis]^.Velocity:=150;
			pMcMoveAbs[E_Axis.Y_Axis]^.Velocity:=150;
			pMcMoveAbs[E_Axis.Z_Axis]^.Velocity:=150;
		ELSE
			pMcMoveAbs[E_Axis.X_Axis]^.Execute:=FALSE;
			pMcMoveAbs[E_Axis.Y_Axis]^.Execute:=FALSE;
			pMcMoveAbs[E_Axis.Z_Axis]^.Execute:=FALSE;
		END_IF;

		IF bCheck1[E_Axis.X_Axis]=TRUE AND bCheck1[E_Axis.Y_Axis]=TRUE AND bCheck1[E_Axis.Z_Axis]=TRUE THEN
			bCheck1[E_Axis.X_Axis]:=FALSE;	
			bCheck1[E_Axis.Y_Axis]:=FALSE;
			bCheck1[E_Axis.Z_Axis]:=FALSE;
			lrDeg:=lrDeg + 1;
			lrBase1[E_Axis.X_Axis]:= stEllipseSettings[iWrittingEllipse].uiVertex * COS(lrDeg*PI/180);
			lrBase1[E_Axis.Y_Axis]:= stEllipseSettings[iWrittingEllipse].uiCoVertex * SIN(lrDeg*PI/180);
			pMcMoveAbsSub[E_Axis.X_Axis]^.Position:=stEllipseSettings[iWrittingEllipse].uiXCenter + lrBase1[E_Axis.X_Axis] * COS(stEllipseSettings[iWrittingEllipse].lrSlopeDeg*PI/180) - lrBase1[E_Axis.Y_Axis] * SIN(stEllipseSettings[iWrittingEllipse].lrSlopeDeg*PI/180);
			pMcMoveAbsSub[E_Axis.Y_Axis]^.Position:=stEllipseSettings[iWrittingEllipse].uiYCenter + lrBase1[E_Axis.X_Axis] * SIN(stEllipseSettings[iWrittingEllipse].lrSlopeDeg*PI/180) + lrBase1[E_Axis.Y_Axis] * COS(stEllipseSettings[iWrittingEllipse].lrSlopeDeg*PI/180);
			
			fbZAxisTPCon1(
				lrX_AxisTP		:=pMcMoveAbsSub[E_Axis.X_Axis]^.Position,
				lrY_AxisTP		:=pMcMoveAbsSub[E_Axis.Y_Axis]^.Position,
				lrZ_AxisTP		:=273-GVL.lrPenFullLength+GVL.lrPenGripLength,
				lrZ_AxisConTP	=>pMcMoveAbsSub[E_Axis.Z_Axis]^.Position
				);

			pMcMoveAbsSub[E_Axis.X_Axis]^.Execute:=TRUE;
			pMcMoveAbsSub[E_Axis.Y_Axis]^.Execute:=TRUE;
			pMcMoveAbsSub[E_Axis.Z_Axis]^.Execute:=TRUE;
			pMcMoveAbsSub[E_Axis.X_Axis]^.Velocity:=150;
			pMcMoveAbsSub[E_Axis.Y_Axis]^.Velocity:=150;
			pMcMoveAbsSub[E_Axis.Z_Axis]^.Velocity:=150;
		ELSE
			pMcMoveAbsSub[E_Axis.X_Axis]^.Execute:=FALSE;
			pMcMoveAbsSub[E_Axis.Y_Axis]^.Execute:=FALSE;
			pMcMoveAbsSub[E_Axis.Z_Axis]^.Execute:=FALSE;
		END_IF;
	
		IF stEllipseSettings[iWrittingEllipse].lrEndDeg < lrDeg THEN
			pMcMoveAbs[E_Axis.X_Axis]^.Execute:=FALSE;
			pMcMoveAbs[E_Axis.Y_Axis]^.Execute:=FALSE;
			pMcMoveAbs[E_Axis.Z_Axis]^.Execute:=FALSE;
			pMcMoveAbsSub[E_Axis.X_Axis]^.Execute:=FALSE;
			pMcMoveAbsSub[E_Axis.Y_Axis]^.Execute:=FALSE;
			pMcMoveAbsSub[E_Axis.Z_Axis]^.Execute:=FALSE;
			eStep:=E_CircleEllipseWriteStep.ZAxisUpPotision;
			iStep:=0;
			lrDeg:=0;
		END_IF;
	
	END_CASE;

E_CircleEllipseWriteStep.ZAxisUpPotision:(*Z軸を持ち上げる、ペンが紙に当たらないように*)

	pMcMoveAbs[E_Axis.Z_Axis]^.Execute:=TRUE;
	pMcMoveAbs[E_Axis.Z_Axis]^.Position:=273-GVL.lrPenFullLength+GVL.lrPenGripLength-50;
	pMcMoveAbs[E_Axis.Z_Axis]^.Velocity:=150;

	IF pMcMoveAbs[E_Axis.Z_Axis]^.Done=TRUE THEN
		eStep:=E_CircleEllipseWriteStep.Check;
		pMcMoveAbs[E_Axis.Z_Axis]^.Execute:=FALSE;
	END_IF;
	
END_CASE
END_METHOD

METHOD FB_init : BOOL
VAR_INPUT
	bInitRetains : BOOL; // if TRUE, the retain variables are initialized (warm start / cold start)
	bInCopyCode : BOOL;  // if TRUE, the instance afterwards gets moved into the copy code (online change)
	rXAxisMcMoveAbs				:REFERENCE TO MC_MoveAbsolute;
	rYAxisMcMoveAbs				:REFERENCE TO MC_MoveAbsolute;
	rZAxisMcMoveAbs				:REFERENCE TO MC_MoveAbsolute;	
	rGripperMcMoveAbs			:REFERENCE TO MC_MoveAbsolute;
	
	rXAxisMcMoveAbsSub			:REFERENCE TO MC_MoveAbsolute;
	rYAxisMcMoveAbsSub			:REFERENCE TO MC_MoveAbsolute;
	rZAxisMcMoveAbsSub			:REFERENCE TO MC_MoveAbsolute;

END_VAR
pMcMoveAbs[E_Axis.X_Axis]:=ADR(rXAxisMcMoveAbs);
pMcMoveAbs[E_Axis.Y_Axis]:=ADR(rYAxisMcMoveAbs);
pMcMoveAbs[E_Axis.Z_Axis]:=ADR(rZAxisMcMoveAbs);
pMcMoveAbs[E_Axis.Gripper]:=ADR(rGripperMcMoveAbs);

pMcMoveAbsSub[E_Axis.X_Axis]:=ADR(rXAxisMcMoveAbsSub);
pMcMoveAbsSub[E_Axis.Y_Axis]:=ADR(rYAxisMcMoveAbsSub);
pMcMoveAbsSub[E_Axis.Z_Axis]:=ADR(rZAxisMcMoveAbsSub);
END_METHOD

PROPERTY iNextProp : INT
SET
iNext:=iNextProp;
END_SET
END_PROPERTY

PROPERTY stCircleSettingsProp :ARRAY[1..32] OF  ST_CircleSettings
SET
stCircleSettings:=stCircleSettingsProp;
END_SET
END_PROPERTY

PROPERTY stEllipseSettingsProp :ARRAY[1..32] OF ST_EllipseSetting
SET
stEllipseSettings:=stEllipseSettingsProp;
END_SET
END_PROPERTY

END_FUNCTION_BLOCK

// ---- POUs/ゴミ箱/FB_Z_Axis_TargetPositionConvert.TcPOU
FUNCTION_BLOCK FB_Z_Axis_TargetPositionConvert
VAR_INPUT
	lrX_AxisTP		:LREAL;	(*X軸のターゲットポジション*)
	lrY_AxisTP		:LREAL;	(*Y軸のターゲットポジション*)
	lrZ_AxisTP		:LREAL;	(*Z軸のターゲットポジション*)
END_VAR
VAR_OUTPUT
	lrZ_AxisConTP	:LREAL;	(*調整後のZ軸のターゲットポジション*)
END_VAR
VAR
	lrXbuf			:LREAL;
	lrYbuf			:LREAL;
END_VAR

	lrXbuf:=GVL.lrXZ_Slope*lrX_AxisTP;
	lrYbuf:=GVL.lrYZ_Slope*lrY_AxisTP;
	
	lrZ_AxisConTP:=lrZ_AxisTP+lrXbuf+lrYbuf;

END_FUNCTION_BLOCK

// ---- POUs/P_MotionWrite.TcPOU
PROGRAM P_MotionWrite
VAR
	eStep				:E_WriteStep:=E_WriteStep.Stay;
	iStep				:INT:=0;
	fbMcMoveAbs			:ARRAY[E_Axis.X_Axis..E_Axis.Gripper] OF MC_MoveAbsolute;
	fbMcMoveAbsSub		:ARRAY[E_Axis.X_Axis..E_Axis.Z_Axis] OF MC_MoveAbsolute;
	fbGripperGripAngle	:FB_Gripper_GripAngle;
	
	stCircleSettings	:ARRAY[1..32] OF ST_CircleSettings;
	stEllipseSettings	:ARRAY[1..32] OF ST_EllipseSetting;

	fbMotionShapeWrite	:FB_MotionShapeWrite(fbMcMoveAbs[E_Axis.X_Axis],
											fbMcMoveAbs[E_Axis.Y_Axis],
											fbMcMoveAbs[E_Axis.Z_Axis],
											fbMcMoveAbs[E_Axis.Gripper],
											fbMcMoveAbsSub[E_Axis.X_Axis],
											fbMcMoveAbsSub[E_Axis.Y_Axis],
											fbMcMoveAbsSub[E_Axis.Z_Axis]);

END_VAR

//WriteMotin実行中か確認
IF eStep<>E_WriteStep.Stay THEN
	
	//McMoveのコマンドアボートをチェック
	IF fbMcMoveAbs[E_Axis.X_Axis].CommandAborted=TRUE
		OR fbMcMoveAbs[E_Axis.Y_Axis].CommandAborted=TRUE
		OR fbMcMoveAbs[E_Axis.Z_Axis].CommandAborted=TRUE
		OR fbMcMoveAbs[E_Axis.Gripper].CommandAborted=TRUE
		OR fbMcMoveAbsSub[E_Axis.X_Axis].CommandAborted=TRUE
		OR fbMcMoveAbsSub[E_Axis.Y_Axis].CommandAborted=TRUE
		OR fbMcMoveAbsSub[E_Axis.Z_Axis].CommandAborted=TRUE THEN
			eStep:=E_WriteStep.CommandAborted;
	END_IF
	
	//McMoveのエラーをチェック
	IF fbMcMoveAbs[E_Axis.X_Axis].Error=TRUE
		OR fbMcMoveAbs[E_Axis.Y_Axis].Error=TRUE
		OR fbMcMoveAbs[E_Axis.Z_Axis].Error=TRUE
		OR fbMcMoveAbs[E_Axis.Gripper].Error=TRUE
		OR fbMcMoveAbsSub[E_Axis.X_Axis].Error=TRUE
		OR fbMcMoveAbsSub[E_Axis.Y_Axis].Error=TRUE
		OR fbMcMoveAbsSub[E_Axis.Z_Axis].Error=TRUE THEN
			eStep:=E_WriteStep.Error;
	END_IF

END_IF
	
CASE eStep OF

E_WriteStep.Stay:(*初期値、bMoveがTrueになったらステップを進める*)

	IF GVL_Motion.bWriteMoveStart=TRUE THEN
		GVL_Motion.bCircleWriteFin:=FALSE;
		GVL_Motion.bEllipseWriteFin:=FALSE;
		GVL_MitsubishiCom.bToWriteMoving:=TRUE;
		eStep:=E_WriteStep.GripperOpen;
	ELSE
		eStep:=E_WriteStep.Stay;
	END_IF;

E_WriteStep.GripperOpen:(*グリッパーを開ける*)
	
	fbMcMoveAbs[E_Axis.Gripper].Execute:=TRUE;
	fbMcMoveAbs[E_Axis.Gripper].Position:=0;
	fbMcMoveAbs[E_Axis.Gripper].Velocity:=150;

	IF fbMcMoveAbs[E_Axis.Gripper].Done=TRUE THEN
		eStep:=E_WriteStep.ZAxixZeroPotision;
		fbMcMoveAbs[E_Axis.Gripper].Execute:=FALSE;
	END_IF;

E_WriteStep.ZAxixZeroPotision:(*Z軸をゼロポジションへ、衝突回避のためにまずZ軸を移動*)

	fbMcMoveAbs[E_Axis.Z_Axis].Execute:=TRUE;
	fbMcMoveAbs[E_Axis.Z_Axis].Position:=0;
	fbMcMoveAbs[E_Axis.Z_Axis].Velocity:=150;

	IF fbMcMoveAbs[E_Axis.Z_Axis].Done=TRUE THEN
		eStep:=E_WriteStep.XYAxixZeroPotision;
		fbMcMoveAbs[E_Axis.Z_Axis].Execute:=FALSE;
	END_IF;

E_WriteStep.XYAxixZeroPotision:(*Z軸移動後に、X,Y軸をゼロポジションへ移動*)

	fbMcMoveAbs[E_Axis.X_Axis].Execute:=TRUE;
	fbMcMoveAbs[E_Axis.Y_Axis].Execute:=TRUE;
	fbMcMoveAbs[E_Axis.X_Axis].Position:=0;
	fbMcMoveAbs[E_Axis.Y_Axis].Position:=0;
	fbMcMoveAbs[E_Axis.X_Axis].Velocity:=150;
	fbMcMoveAbs[E_Axis.Y_Axis].Velocity:=150;
	
	IF fbMcMoveAbs[E_Axis.X_Axis].Done=TRUE AND fbMcMoveAbs[E_Axis.Y_Axis].Done=TRUE THEN
		eStep:=E_WriteStep.PenGripp;
		fbMcMoveAbs[E_Axis.X_Axis].Execute:=FALSE;
		fbMcMoveAbs[E_Axis.Y_Axis].Execute:=FALSE;
	END_IF;

E_WriteStep.PenGripp:(*ペンを掴む*)

	CASE iStep OF
	0:(*何もしない*)
		iStep:=1;
	
	1:(*ペンを掴む高さに移動*)
		fbMcMoveAbs[E_Axis.Z_Axis].Execute:=TRUE;
		fbMcMoveAbs[E_Axis.Z_Axis].Position:=205.0-GVL.lrPenHalfLength+GVL.lrPenGripLength;
		fbMcMoveAbs[E_Axis.Z_Axis].Velocity:=150;

		IF fbMcMoveAbs[E_Axis.Z_Axis].Done=TRUE THEN
			iStep:=2;
			fbMcMoveAbs[E_Axis.Z_Axis].Execute:=FALSE;
		END_IF;
	
	2:(*グリッパーを閉じてペンを掴む*)
		fbMcMoveAbs[E_Axis.Gripper].Execute:=TRUE;
		
		fbGripperGripAngle(
			lrPenDiameter:=GVL.lrPenDiameter,
			lrGripAngle=>fbMcMoveAbs[E_Axis.Gripper].Position
			);

		fbMcMoveAbs[E_Axis.Gripper].Velocity:=150;
	
		IF fbMcMoveAbs[E_Axis.Gripper].Done=TRUE THEN
			iStep:=3;
			fbMcMoveAbs[E_Axis.Gripper].Execute:=FALSE;
		END_IF;
	
	3:(*Z軸をゼロポジションへ戻す*)
		fbMcMoveAbs[E_Axis.Z_Axis].Execute:=TRUE;
		fbMcMoveAbs[E_Axis.Z_Axis].Position:=0;
		fbMcMoveAbs[E_Axis.Z_Axis].Velocity:=150;
	
		IF fbMcMoveAbs[E_Axis.Z_Axis].Done=TRUE THEN
			eStep:=E_WriteStep.Write;
			fbMcMoveAbs[E_Axis.Z_Axis].Execute:=FALSE;
			iStep:=0;
		END_IF;
	
	END_CASE;

E_WriteStep.Write:(*図形を書いていく*)
	CASE iStep OF
	0:
		iStep:=1;
	
	1:
		fbMotionShapeWrite.stCircleSettingsProp:=stCircleSettings;
		fbMotionShapeWrite.stEllipseSettingsProp:=stEllipseSettings;
		
		fbMotionShapeWrite.bStartProp:=TRUE;
		
		IF fbMotionShapeWrite.bEndProp=TRUE THEN
			fbMotionShapeWrite.bStartProp:=FALSE;
			fbMotionShapeWrite.bEndProp:=FALSE;
			iStep:=2;
		END_IF
		
		fbMotionShapeWrite();
		
	2:
		eStep:=E_WriteStep.ZAxixZeroPotision2;
		iStep:=0;
		
	END_CASE

E_WriteStep.ZAxixZeroPotision2:(*Z軸をゼロポジションへ、衝突回避のためにまずZ軸を移動*)

	fbMcMoveAbs[E_Axis.Z_Axis].Execute:=TRUE;
	fbMcMoveAbs[E_Axis.Z_Axis].Position:=0;
	fbMcMoveAbs[E_Axis.Z_Axis].Velocity:=150;

	IF fbMcMoveAbs[E_Axis.Z_Axis].Done=TRUE THEN
		eStep:=E_WriteStep.XYAxixZeroPotision2;
		fbMcMoveAbs[E_Axis.Z_Axis].Execute:=FALSE;
	END_IF;
	
E_WriteStep.XYAxixZeroPotision2:(*Z軸移動後に、X,Y軸をゼロポジションへ移動*)

	fbMcMoveAbs[E_Axis.X_Axis].Execute:=TRUE;
	fbMcMoveAbs[E_Axis.Y_Axis].Execute:=TRUE;
	fbMcMoveAbs[E_Axis.X_Axis].Position:=0;
	fbMcMoveAbs[E_Axis.Y_Axis].Position:=0;
	fbMcMoveAbs[E_Axis.X_Axis].Velocity:=150;
	fbMcMoveAbs[E_Axis.Y_Axis].Velocity:=150;
	
	IF fbMcMoveAbs[E_Axis.X_Axis].Done=TRUE AND fbMcMoveAbs[E_Axis.Y_Axis].Done=TRUE THEN
		eStep:=E_WriteStep.PenRelease;
		fbMcMoveAbs[E_Axis.X_Axis].Execute:=FALSE;
		fbMcMoveAbs[E_Axis.Y_Axis].Execute:=FALSE;
	END_IF;

E_WriteStep.PenRelease:(*ペンをリリースする*)

	CASE iStep OF
	0:
		iStep:=1;
		
	1:
		fbMcMoveAbs[E_Axis.Z_Axis].Execute:=TRUE;
		fbMcMoveAbs[E_Axis.Z_Axis].Position:=205.0-GVL.lrPenHalfLength+GVL.lrPenGripLength;
		
		IF fbMcMoveAbs[E_Axis.Z_Axis].Done=TRUE THEN
			fbMcMoveAbs[E_Axis.Z_Axis].Execute:=FALSE;
			iStep:=2;
		END_IF;
	
	2:
		fbMcMoveAbs[E_Axis.Gripper].Execute:=TRUE;
		fbMcMoveAbs[E_Axis.Gripper].Position:=0;
	
		IF fbMcMoveAbs[E_Axis.Gripper].Done=TRUE THEN
			fbMcMoveAbs[E_Axis.Gripper].Execute:=FALSE;
			iStep:=3;
		END_IF;
	
	3:
		fbMcMoveAbs[E_Axis.Z_Axis].Execute:=TRUE;
		fbMcMoveAbs[E_Axis.Z_Axis].Position:=0;

		IF fbMcMoveAbs[E_Axis.Z_Axis].Done=TRUE THEN
			eStep:=E_WriteStep.Stay;
			fbMcMoveAbs[E_Axis.Z_Axis].Execute:=FALSE;
			iStep:=0;
			GVL_MitsubishiCom.bToWriteMoving:=FALSE;
		END_IF;
	
	END_CASE;
	
E_WriteStep.CommandAborted://McMoveコマンドアボート時の処理	

	iStep:=0;
	fbMcMoveAbs[E_Axis.X_Axis].Execute:=FALSE;
	fbMcMoveAbs[E_Axis.Y_Axis].Execute:=FALSE;
	fbMcMoveAbs[E_Axis.Z_Axis].Execute:=FALSE;
	fbMcMoveAbs[E_Axis.Gripper].Execute:=FALSE;

	fbMcMoveAbsSub[E_Axis.X_Axis].Execute:=FALSE;
	fbMcMoveAbsSub[E_Axis.Y_Axis].Execute:=FALSE;
	fbMcMoveAbsSub[E_Axis.Z_Axis].Execute:=FALSE;
	
	GVL_MitsubishiCom.bToAutoMoveResetting:=FALSE;

	IF fbMcMoveAbs[E_Axis.X_Axis].CommandAborted=FALSE
		AND fbMcMoveAbs[E_Axis.Y_Axis].CommandAborted=FALSE
		AND fbMcMoveAbs[E_Axis.Z_Axis].CommandAborted=FALSE
		AND fbMcMoveAbs[E_Axis.Gripper].CommandAborted=FALSE
		AND fbMcMoveAbsSub[E_Axis.X_Axis].CommandAborted=FALSE
		AND fbMcMoveAbsSub[E_Axis.Y_Axis].CommandAborted=FALSE
		AND fbMcMoveAbsSub[E_Axis.Z_Axis].CommandAborted=FALSE THEN
			eStep:=E_WriteStep.Reset;
	END_IF

E_WriteStep.Error://McMoveエラー時の処理	

	iStep:=0;
	fbMcMoveAbs[E_Axis.X_Axis].Execute:=FALSE;
	fbMcMoveAbs[E_Axis.Y_Axis].Execute:=FALSE;
	fbMcMoveAbs[E_Axis.Z_Axis].Execute:=FALSE;
	fbMcMoveAbs[E_Axis.Gripper].Execute:=FALSE;

	fbMcMoveAbsSub[E_Axis.X_Axis].Execute:=FALSE;
	fbMcMoveAbsSub[E_Axis.Y_Axis].Execute:=FALSE;
	fbMcMoveAbsSub[E_Axis.Z_Axis].Execute:=FALSE;
	
	GVL_MitsubishiCom.bToAutoMoveResetting:=FALSE;

	if fbMcMoveAbs[E_Axis.X_Axis].Error=FALSE
		AND fbMcMoveAbs[E_Axis.Y_Axis].Error=FALSE
		AND fbMcMoveAbs[E_Axis.Z_Axis].Error=FALSE
		AND fbMcMoveAbs[E_Axis.Gripper].Error=FALSE
		AND fbMcMoveAbsSub[E_Axis.X_Axis].Error=FALSE
		AND fbMcMoveAbsSub[E_Axis.Y_Axis].Error=FALSE
		AND fbMcMoveAbsSub[E_Axis.Z_Axis].Error=FALSE THEN
			eStep:=E_WriteStep.Reset;
	END_IF	
	
E_WriteStep.Reset://McMoveのコマンドアボートorエラー後のリセット動作

	CASE iStep OF

	0:
		IF GVL_MitsubishiCom.bFromAutoMoveReset=TRUE AND MAIN.fb3AxisRobot.fbMachineState.bStopMachine=FALSE THEN
			GVL_MitsubishiCom.bToAutoMoveResetting:=TRUE;
			iStep:=1;
			//FB_MotionShapeWriteのリセット
			fbMotionShapeWrite.iNextProp:=0;
		END_IF

	1:
		fbMcMoveAbs[E_Axis.Gripper].Execute:=TRUE;
		fbMcMoveAbs[E_Axis.Gripper].Position:=0;
		fbMcMoveAbs[E_Axis.Gripper].Velocity:=150;

		IF fbMcMoveAbs[E_Axis.Gripper].Done=TRUE THEN
			iStep:=2;
			fbMcMoveAbs[E_Axis.Gripper].Execute:=FALSE;
		END_IF;

	2:
		fbMcMoveAbs[E_Axis.Z_Axis].Execute:=TRUE;
		fbMcMoveAbs[E_Axis.Z_Axis].Position:=0;
		fbMcMoveAbs[E_Axis.Z_Axis].Velocity:=150;

		IF fbMcMoveAbs[E_Axis.Z_Axis].Done=TRUE THEN
			iStep:=3;
			fbMcMoveAbs[E_Axis.Z_Axis].Execute:=FALSE;
		END_IF;

	3:
		fbMcMoveAbs[E_Axis.X_Axis].Execute:=TRUE;
		fbMcMoveAbs[E_Axis.Y_Axis].Execute:=TRUE;
		fbMcMoveAbs[E_Axis.X_Axis].Position:=0;
		fbMcMoveAbs[E_Axis.Y_Axis].Position:=0;
		fbMcMoveAbs[E_Axis.X_Axis].Velocity:=150;
		fbMcMoveAbs[E_Axis.Y_Axis].Velocity:=150;

		IF fbMcMoveAbs[E_Axis.X_Axis].Done=TRUE AND fbMcMoveAbs[E_Axis.Y_Axis].Done=TRUE THEN
			fbMcMoveAbs[E_Axis.X_Axis].Execute:=FALSE;
			fbMcMoveAbs[E_Axis.Y_Axis].Execute:=FALSE;
			iStep:=0;
			eStep:=E_WriteStep.Stay;

			GVL_MitsubishiCom.bToWriteMoving:=FALSE;
			GVL_MitsubishiCom.bToAutoMoveResetting:=FALSE;
		END_IF;

	END_CASE
	
END_CASE;

	aMotion();

ACTION aMotion:
//各軸とグリッパーの駆動用
	//メイン
	fbMcMoveAbs[E_Axis.X_Axis](
		Axis			:=GVL_Axis.stAxis[E_Axis.X_Axis],
		BufferMode		:=MC_BlendingNext,
	);

	fbMcMoveAbs[E_Axis.Y_Axis](
		Axis			:=GVL_Axis.stAxis[E_Axis.Y_Axis],
		BufferMode		:=MC_BlendingNext,
	);

	fbMcMoveAbs[E_Axis.Z_Axis](
		Axis			:=GVL_Axis.stAxis[E_Axis.Z_Axis],
		BufferMode		:=MC_BlendingNext,
	);
	
	fbMcMoveAbs[E_Axis.Gripper](
		Axis			:=GVL_Axis.stAxis[E_Axis.Gripper],
		BufferMode		:=MC_BlendingNext,
	);
	
	//ここからサブ、サブはグリッパー無し
	fbMcMoveAbsSub[E_Axis.X_Axis](
		Axis			:=GVL_Axis.stAxis[E_Axis.X_Axis],
		BufferMode		:=MC_BlendingNext,
	);

	fbMcMoveAbsSub[E_Axis.Y_Axis](
		Axis			:=GVL_Axis.stAxis[E_Axis.Y_Axis],
		BufferMode		:=MC_BlendingNext,
	);

	fbMcMoveAbsSub[E_Axis.Z_Axis](
		Axis			:=GVL_Axis.stAxis[E_Axis.Z_Axis],
		BufferMode		:=MC_BlendingNext,
	);
END_ACTION

END_PROGRAM

// ---- POUs/ゴミ箱/FB_Gripper_GripAngle.TcPOU
FUNCTION_BLOCK FB_Gripper_GripAngle
VAR_INPUT
	lrPenDiameter	:lREAL;(*ペンの直径 単位mm*)
END_VAR
VAR_OUTPUT
	lrGripAngle		:LREAL;(*グリップする角度*)
END_VAR
VAR
	lrd				:LREAL:=6.000;(*アタッチメントの直径［mm］*)
	lrr				:LREAL:=6.400;(*アタッチメントの回転半径［mm］*)
	lrA				:LREAL;
	lrB				:LREAL;
END_VAR

	lrA:=EXPT((lrPenDiameter+lrd)/2,2)-EXPT(9.05,2)-EXPT(lrr,2);
	lrB:=2*9.05*lrr;

	IF -1<lrA/lrB AND lrA/lrB<1 THEN
		lrGripAngle:=180/PI*ACOS(lrA/lrB);
	END_IF;

END_FUNCTION_BLOCK

// ---- POUs/ゴミ箱/FB_3AxisAbs.TcPOU
FUNCTION_BLOCK FB_3AxisAbs
VAR_INPUT
END_VAR
VAR
	_bAxisError				:ARRAY[E_Axis.X_Axis..E_Axis.Gripper] OF BOOL;				//各軸Error
	nAxisErrorID			:ARRAY[E_Axis.X_Axis..E_Axis.Gripper] OF UDINT;				//各軸Error ID
	_bAxisMoving			:ARRAY[E_Axis.X_Axis..E_Axis.Gripper] OF BOOL;				//各軸moving
	_fAxisActPos			:ARRAY[E_Axis.X_Axis..E_Axis.Gripper] OF LREAL;				//各軸Actual Position
	
	_bAxisEnable			:ARRAY[E_Axis.X_Axis..E_Axis.Gripper] OF BOOL;				//各軸PoerON
	_bResetDone				:ARRAY[E_Axis.X_Axis..E_Axis.Gripper] OF BOOL;				//各軸リセット完了
	_bHaltDone				:ARRAY[E_Axis.X_Axis..E_Axis.Gripper] OF BOOL;				//各軸一時停止完了
	_bStopDone				:ARRAY[E_Axis.X_Axis..E_Axis.Gripper] OF BOOL;				//各軸停止完了





	

END_VAR

//---なし---

METHOD AbsMove
VAR_INPUT
	eAxis			:E_Axis;
	bMove			:BOOL;
	fTargetPos		:LREAL;
	fTargetVelo		:LREAL;
END_VAR
CASE eAxis OF
	E_Axis.X_Axis:
		fbXAxis.fTargetPosition:=fTargetPos;
		fbXAxis.fTargetVelocity:=fTargetVelo;
		fbXAxis.MoveAbsolute(bMove:=bMove);

	E_Axis.Y_Axis:
		fbYAxis.fTargetPosition:=fTargetPos;
		fbYAxis.fTargetVelocity:=fTargetVelo;
		fbYAxis.MoveAbsolute(bMove:=bMove);
	
	E_Axis.Z_Axis:
		fbZAxis.fTargetPosition:=fTargetPos;
		fbZAxis.fTargetVelocity:=fTargetVelo;
		fbZAxis.MoveAbsolute(bMove:=bMove);
		
	E_Axis.Gripper:
		fbGripper.fTargetPosition:=fTargetPos;
		fbGripper.fTargetVelocity:=fTargetVelo;
		fbGripper.MoveAbsolute(bMove:=bMove);
	
END_CASE
END_METHOD

METHOD bAxisError : BOOL
VAR_INPUT
	eAxis	:E_Axis;
END_VAR
bAxisError:=_bAxisError[eAxis];
END_METHOD

METHOD bAxisMoving : BOOL
VAR_INPUT
	eAxis	:E_Axis;
END_VAR
bAxisMoving:=_bAxisMoving[eAxis];
END_METHOD

PROPERTY bEnable : BOOL
GET
bEnable:=_bAxisEnable[E_Axis.X_Axis] AND _bAxisEnable[E_Axis.Y_Axis] AND _bAxisEnable[E_Axis.Z_Axis] AND _bAxisEnable[E_Axis.Gripper];
END_GET
END_PROPERTY

PROPERTY bError : BOOL
GET
bError:=_bAxisError[E_Axis.X_Axis] or _bAxisError[E_Axis.Y_Axis] or _bAxisError[E_Axis.Z_Axis] or _bAxisError[E_Axis.Gripper];
END_GET
END_PROPERTY

PROPERTY bHaltDone : BOOL
GET
bHaltDone:=_bHaltDone[E_Axis.X_Axis] AND _bHaltDone[E_Axis.Y_Axis] AND _bHaltDone[E_Axis.Z_Axis] AND _bHaltDone[E_Axis.Gripper];
END_GET
END_PROPERTY

PROPERTY bMoving : BOOL
GET
bMoving:=_bAxisMoving[E_Axis.X_Axis] or _bAxisMoving[E_Axis.Y_Axis] or _bAxisMoving[E_Axis.Z_Axis] or _bAxisMoving[E_Axis.Gripper];
END_GET
END_PROPERTY

PROPERTY bResetDone : BOOL
GET
bResetDone:=_bResetDone[E_Axis.X_Axis] AND _bResetDone[E_Axis.Y_Axis] AND _bResetDone[E_Axis.Z_Axis] AND _bResetDone[E_Axis.Gripper];
END_GET
END_PROPERTY

PROPERTY bStopDone : BOOL
GET
bStopDone:=_bStopDone[E_Axis.X_Axis] AND _bStopDone[E_Axis.Y_Axis] AND _bStopDone[E_Axis.Z_Axis] AND _bStopDone[E_Axis.Gripper];
END_GET
END_PROPERTY

METHOD fAxisActPos : LREAL
VAR_INPUT
	eAxis	:E_Axis;
END_VAR
fAxisActPos:=_fAxisActPos[eAxis];
END_METHOD

METHOD Halt
VAR_INPUT
	bHalt		: BOOL;
END_VAR
// =========================================================
// Halting axis

	fbXAxis.Halt(bDriveHalt:= bHalt);
	fbYAxis.Halt(bDriveHalt:= bHalt);
	fbZAxis.Halt(bDriveHalt:= bHalt);
	fbGripper.Halt(bDriveHalt:= bHalt);

	_bHaltDone[E_Axis.X_Axis]:=fbXAxis.bStateHaltDone;
	_bHaltDone[E_Axis.Y_Axis]:=fbYAxis.bStateHaltDone;
	_bHaltDone[E_Axis.Z_Axis]:=fbZAxis.bStateHaltDone;
	_bHaltDone[E_Axis.Gripper]:=fbGripper.bStateHaltDone;

// =========================================================
END_METHOD

METHOD Homing: BOOL
VAR_INPUT
	bHome						:BOOL;
END_VAR
IF bHome=TRUE THEN
	fbXAxis.fTargetPosition:=0;
	fbYAxis.fTargetPosition:=0;
	fbZAxis.fTargetPosition:=0;
	fbGripper.fTargetPosition:=0;
	
	fbXAxis.fTargetVelocity:=50;
	fbYAxis.fTargetVelocity:=50;
	fbZAxis.fTargetVelocity:=50;
	fbGripper.fTargetVelocity:=100;
END_IF

fbXAxis.MoveAbsolute(bMove:=bHome);
fbYAxis.MoveAbsolute(bMove:=bHome);
fbZAxis.MoveAbsolute(bMove:=bHome);
fbGripper.MoveAbsolute(bMove:=bHome);


IF bHome=TRUE AND bMoving=TRUE THEN
	Homing:=TRUE;
ELSIF bMoving=FALSE THEN
	Homing:=FALSE;
END_IF
END_METHOD

METHOD Jog
VAR_INPUT
	eAxis			:E_Axis;
	bMove			:BOOL;
	fTargetPos		:LREAL;
	fTargetVelo		:LREAL;
END_VAR
//立下りエッジを取得	
fbJogFEdge[eAxis](CLK:=bMove,Q=>);

CASE eAxis OF
	E_Axis.X_Axis:
		fbXAxis.fTargetPosition:=fTargetPos;
		fbXAxis.fTargetVelocity:=fTargetVelo;
		fbXAxis.MoveAbsolute(bMove:=bMove);
		fbXAxis.Halt(bDriveHalt:=fbJogFEdge[eAxis].Q);

	E_Axis.Y_Axis:
		fbYAxis.fTargetPosition:=fTargetPos;
		fbYAxis.fTargetVelocity:=fTargetVelo;
		fbYAxis.MoveAbsolute(bMove:=bMove);
		fbYAxis.Halt(bDriveHalt:=fbJogFEdge[eAxis].Q);
	
	E_Axis.Z_Axis:
		fbZAxis.fTargetPosition:=fTargetPos;
		fbZAxis.fTargetVelocity:=fTargetVelo;
		fbZAxis.MoveAbsolute(bMove:=bMove);
		fbZAxis.Halt(bDriveHalt:=fbJogFEdge[eAxis].Q);
		
	E_Axis.Gripper:
		fbGripper.fTargetPosition:=fTargetPos;
		fbGripper.fTargetVelocity:=fTargetVelo;
		fbGripper.MoveAbsolute(bMove:=bMove);
		fbGripper.Halt(bDriveHalt:=fbJogFEdge[eAxis].Q);
	
END_CASE
END_METHOD

METHOD Power
VAR_INPUT
	bAxisEnable				: BOOL;			// Enable of axis
END_VAR

	
	

	_bAxisError[E_Axis.X_Axis]	:=fbXAxis.bStateError;
	nAxisErrorID[E_Axis.X_Axis]	:=fbXAxis.nStateErrorID;
	_bAxisMoving[E_Axis.X_Axis]	:=fbXAxis.bStateMoving;
	_fAxisActPos[E_Axis.X_Axis]	:=fbXAxis.fStateActPos;

	
	
	_bAxisError[E_Axis.Y_Axis]	:=fbYAxis.bStateError;
	nAxisErrorID[E_Axis.Y_Axis]	:=fbYAxis.nStateErrorID;
	_bAxisMoving[E_Axis.Y_Axis]	:=fbYAxis.bStateMoving;
	_fAxisActPos[E_Axis.Y_Axis]	:=fbYAxis.fStateActPos;

	
		
	_bAxisError[E_Axis.Z_Axis]	:=fbZAxis.bStateError;
	nAxisErrorID[E_Axis.Z_Axis]	:=fbZAxis.nStateErrorID;
	_bAxisMoving[E_Axis.Z_Axis]	:=fbZAxis.bStateMoving;
	_fAxisActPos[E_Axis.Z_Axis]	:=fbZAxis.fStateActPos;
	
	
		
	_bAxisError[E_Axis.Gripper]	:=fbGripper.bStateError;
	nAxisErrorID[E_Axis.Gripper]:=fbGripper.nStateErrorID;
	_bAxisMoving[E_Axis.Gripper]:=fbGripper.bStateMoving;
	_fAxisActPos[E_Axis.Gripper]:=fbGripper.fStateActPos;
END_METHOD

METHOD Reset : BOOL
VAR_INPUT
	bReset		: BOOL;
END_VAR
// =========================================================
// Resetting axis

	fbXAxis.Reset(bDriveReset := bReset);
	fbYAxis.Reset(bDriveReset := bReset);
	fbZAxis.Reset(bDriveReset := bReset);
	fbGripper.Reset(bDriveReset := bReset);
	
	_bResetDone[E_Axis.X_Axis]:=fbXAxis.bStateResetDone;
	_bResetDone[E_Axis.Y_Axis]:=fbYAxis.bStateResetDone;
	_bResetDone[E_Axis.Z_Axis]:=fbZAxis.bStateResetDone;
	_bResetDone[E_Axis.Gripper]:=fbGripper.bStateResetDone;

// =========================================================
END_METHOD

METHOD Stop
VAR_INPUT
	bStop		: BOOL;	
END_VAR
// =========================================================
// Stopping axis

	fbXAxis.Stop(bDriveStop := bStop);
	fbYAxis.Stop(bDriveStop := bStop);
	fbZAxis.Stop(bDriveStop := bStop);
	fbGripper.Stop(bDriveStop := bStop);
	
	_bStopDone[E_Axis.X_Axis]:=fbXAxis.bStateStopDone;
	_bStopDone[E_Axis.Y_Axis]:=fbYAxis.bStateStopDone;
	_bStopDone[E_Axis.Z_Axis]:=fbZAxis.bStateStopDone;
	_bStopDone[E_Axis.Gripper]:=fbGripper.bStateStopDone;
		
// =========================================================
END_METHOD

END_FUNCTION_BLOCK

// ---- POUs/ゴミ箱/FB_DiagnosisEtherCAT.TcPOU
FUNCTION_BLOCK FB_DiagnosisEtherCAT
VAR
	uiDevState 			AT%I*	:UINT;
	uiFrmState 			AT%I*	:ARRAY[0..uiMaxFrmNumber] OF UINT;
	uiFrmWcState 		AT%I*	:ARRAY[0..uiMaxFrmNumber] OF UINT;
	uiSlaveCount 		AT%I*	:UINT;
	uiCfgSlaveCount 	AT%I*	:UINT;

	sDevStateStatus				:STRING(255);	
	sFrmStateStatus				:STRING(255);
	sFrmWcStateStatus			:STRING(255);
END_VAR
VAR CONSTANT
	uiMaxFrmNumber				:UINT :=2 ;
END_VAR

METHOD DevState_Diagnosis : BOOL
VAR_INPUT
END_VAR
//デバイスの状態チェック、エラーは複数発生する可能性があるので全bitチェック
IF uiDevState.0 THEN
	sDevStateStatus:= 'Link error. ';
ELSE
	sDevStateStatus:= '';
END_IF
IF uiDevState.1 THEN
	sDevStateStatus:= CONCAT( sDevStateStatus, 'I/O locked after link error (I/O reset required). ');
ELSE
	sDevStateStatus:= CONCAT( sDevStateStatus, '');
END_IF
IF uiDevState.2 THEN
	sDevStateStatus:= CONCAT( sDevStateStatus, 'Link error (redundancy adapter). ');
ELSE
	sDevStateStatus:= CONCAT( sDevStateStatus, '');
END_IF
IF uiDevState.3 THEN
	sDevStateStatus:= CONCAT( sDevStateStatus, 'Missing one frame (redundancy mode). ');
ELSE
	sDevStateStatus:= CONCAT( sDevStateStatus, '');
END_IF
IF uiDevState.4 THEN
	sDevStateStatus:= CONCAT( sDevStateStatus, 'Out of send resources (I/O reset required). ');
ELSE
	sDevStateStatus:= CONCAT( sDevStateStatus, '');
END_IF
IF uiDevState.5 THEN
	sDevStateStatus:= CONCAT( sDevStateStatus, 'Watchdog triggered. ');
ELSE
	sDevStateStatus:= CONCAT( sDevStateStatus, '');
END_IF
IF uiDevState.6 THEN
	sDevStateStatus:= CONCAT( sDevStateStatus, 'Ethernet driver (miniport not found). ');
ELSE
	sDevStateStatus:= CONCAT( sDevStateStatus, '');
END_IF
IF uiDevState.7 THEN
	sDevStateStatus:= CONCAT( sDevStateStatus, 'I/O reset active. ');
ELSE
	sDevStateStatus:= CONCAT( sDevStateStatus, '');
END_IF
IF uiDevState.8 THEN
	sDevStateStatus:= CONCAT( sDevStateStatus, 'At least one device in INIT state. ');
ELSE
	sDevStateStatus:= CONCAT( sDevStateStatus, '');
END_IF
IF uiDevState.9 THEN
	sDevStateStatus:= CONCAT( sDevStateStatus, 'At least one device in PRE-OP state. ');
ELSE
	sDevStateStatus:= CONCAT( sDevStateStatus, '');
END_IF
IF uiDevState.10 THEN
	sDevStateStatus:= CONCAT( sDevStateStatus, 'At least one device in SAFE-OP state. ');
ELSE
	sDevStateStatus:= CONCAT( sDevStateStatus, '');
END_IF
IF uiDevState.11 THEN
	sDevStateStatus:= CONCAT( sDevStateStatus, 'At least on device indicates an error state. ');
ELSE
	sDevStateStatus:= CONCAT( sDevStateStatus, '');
END_IF
IF uiDevState.12 THEN
	sDevStateStatus:= CONCAT( sDevStateStatus, 'DC not in sync. ');
ELSE
	sDevStateStatus:= CONCAT( sDevStateStatus, '');
END_IF


IF sDevStateStatus= '' THEN
	DevState_Diagnosis:= TRUE;
ELSE
	DevState_Diagnosis:= FALSE;
END_IF
END_METHOD

METHOD FrmState_Diagnosis : BOOL
VAR_INPUT
	iFrmNumber		:INT;
END_VAR
//フレームの状態チェック、エラーは複数発生する可能性があるので全bitチェック
IF (uiFrmState[iFrmNumber] < 32768 AND uiFrmState[iFrmNumber] <>0) OR uiFrmState[iFrmNumber] > 32768 THEN

	IF uiFrmState[iFrmNumber].0 THEN
		sFrmStateStatus:= '1. ';
	ELSE
		sFrmStateStatus:= '';
	END_IF
	IF uiFrmState[iFrmNumber].1 THEN
		sFrmStateStatus:= CONCAT( sFrmStateStatus, '2. ');
	ELSE
		sFrmStateStatus:= CONCAT( sFrmStateStatus, '');
	END_IF
	IF uiFrmState[iFrmNumber].2 THEN
		sFrmStateStatus:= CONCAT( sFrmStateStatus, '3. ');
	ELSE
		sFrmStateStatus:= CONCAT( sFrmStateStatus, '');
	END_IF
	IF uiFrmState[iFrmNumber].3 THEN
		sFrmStateStatus:= CONCAT( sFrmStateStatus, '4. ');
	ELSE
		sFrmStateStatus:= CONCAT( sFrmStateStatus, '');
	END_IF
	IF uiFrmState[iFrmNumber].4 THEN
		sFrmStateStatus:= CONCAT( sFrmStateStatus, '5. ');
	ELSE
		sFrmStateStatus:= CONCAT( sFrmStateStatus, '');
	END_IF
	IF uiFrmState[iFrmNumber].5 THEN
		sFrmStateStatus:= CONCAT( sFrmStateStatus, '6. ');
	ELSE
		sFrmStateStatus:= CONCAT( sFrmStateStatus, '');
	END_IF
	IF uiFrmState[iFrmNumber].6 THEN
		sFrmStateStatus:= CONCAT( sFrmStateStatus, '7. ');
	ELSE
		sFrmStateStatus:= CONCAT( sFrmStateStatus, '');
	END_IF
	IF uiFrmState[iFrmNumber].7 THEN
		sFrmStateStatus:= CONCAT( sFrmStateStatus, '8. ');
	ELSE
		sFrmStateStatus:= CONCAT( sFrmStateStatus, '');
	END_IF
	IF uiFrmState[iFrmNumber].8 THEN
		sFrmStateStatus:= CONCAT( sFrmStateStatus, '9. ');
	ELSE
		sFrmStateStatus:= CONCAT( sFrmStateStatus, '');
	END_IF
	IF uiFrmState[iFrmNumber].9 THEN
		sFrmStateStatus:= CONCAT( sFrmStateStatus, '10. ');
	ELSE
		sFrmStateStatus:= CONCAT( sFrmStateStatus, '');
	END_IF
	IF uiFrmState[iFrmNumber].10 THEN
		sFrmStateStatus:= CONCAT( sFrmStateStatus, '11. ');
	ELSE
		sFrmStateStatus:= CONCAT( sFrmStateStatus, '');
	END_IF
	IF uiFrmState[iFrmNumber].11 THEN
		sFrmStateStatus:= CONCAT( sFrmStateStatus, '12. ');
	ELSE
		sFrmStateStatus:= CONCAT( sFrmStateStatus, '');
	END_IF
	IF uiFrmState[iFrmNumber].12 THEN
		sFrmStateStatus:= CONCAT( sFrmStateStatus, '13. ');
	ELSE
		sFrmStateStatus:= CONCAT( sFrmStateStatus, '');
	END_IF
	IF uiFrmState[iFrmNumber].13 THEN
		sFrmStateStatus:= CONCAT( sFrmStateStatus, '14. ');
	ELSE
		sFrmStateStatus:= CONCAT( sFrmStateStatus, '');
	END_IF
	IF uiFrmState[iFrmNumber].14 THEN
		sFrmStateStatus:= CONCAT( sFrmStateStatus, '15. ');
	ELSE
		sFrmStateStatus:= CONCAT( sFrmStateStatus, '');
	END_IF

	sFrmStateStatus:=CONCAT(sFrmStateStatus, 'EtherCAT command not sent (NOP requested). ');

ELSIF uiFrmState[iFrmNumber]= 0 THEN
	sFrmStateStatus:= '';
END_IF

IF uiFrmState[iFrmNumber].15 THEN
	sFrmStateStatus:=  'Complete frame not sent. ';
ELSE
	sFrmStateStatus:= CONCAT( sFrmStateStatus, '');
END_IF


IF sFrmStateStatus= '' THEN
	FrmState_Diagnosis:= TRUE;
ELSE
	FrmState_Diagnosis:= FALSE;
END_IF
END_METHOD

METHOD FrmWcState_Diagnosis : BOOL
VAR_INPUT
	iFrmNumber		:INT;
END_VAR
//サイクリックフレームごとのワーキングカウンターチェック、エラーは複数発生する可能性があるので全bitチェック
IF (uiFrmWcState[iFrmNumber] < 32768 AND uiFrmWcState[iFrmNumber]<>0) OR uiFrmWcState[iFrmNumber]>32768  THEN
	sFrmWcStateStatus:= 'Wrong working counter of ';

	IF uiFrmWcState[iFrmNumber].0 THEN
		sFrmWcStateStatus:= CONCAT( sFrmWcStateStatus, '1. ');
	ELSE
		sFrmWcStateStatus:= CONCAT( sFrmWcStateStatus, '');
	END_IF
	IF uiFrmWcState[iFrmNumber].1 THEN
		sFrmWcStateStatus:= CONCAT( sFrmWcStateStatus, '2. ');
	ELSE
		sFrmWcStateStatus:= CONCAT( sFrmWcStateStatus, '');
	END_IF
	IF uiFrmWcState[iFrmNumber].2 THEN
		sFrmWcStateStatus:= CONCAT( sFrmWcStateStatus, '3. ');
	ELSE
		sFrmWcStateStatus:= CONCAT( sFrmWcStateStatus, '');
	END_IF
	IF uiFrmWcState[iFrmNumber].3 THEN
		sFrmWcStateStatus:= CONCAT( sFrmWcStateStatus, '4. ');
	ELSE
		sFrmWcStateStatus:= CONCAT( sFrmWcStateStatus, '');
	END_IF
	IF uiFrmWcState[iFrmNumber].4 THEN
		sFrmWcStateStatus:= CONCAT( sFrmWcStateStatus, '5. ');
	ELSE
		sFrmWcStateStatus:= CONCAT( sFrmWcStateStatus, '');
	END_IF
	IF uiFrmWcState[iFrmNumber].5 THEN
		sFrmWcStateStatus:= CONCAT( sFrmWcStateStatus, '6. ');
	ELSE
		sFrmWcStateStatus:= CONCAT( sFrmWcStateStatus, '');
	END_IF
	IF uiFrmWcState[iFrmNumber].6 THEN
		sFrmWcStateStatus:= CONCAT( sFrmWcStateStatus, '7. ');
	ELSE
		sFrmWcStateStatus:= CONCAT( sFrmWcStateStatus, '');
	END_IF
	IF uiFrmWcState[iFrmNumber].7 THEN
		sFrmWcStateStatus:= CONCAT( sFrmWcStateStatus, '8. ');
	ELSE
		sFrmWcStateStatus:= CONCAT( sFrmWcStateStatus, '');
	END_IF
	IF uiFrmWcState[iFrmNumber].8 THEN
		sFrmWcStateStatus:= CONCAT( sFrmWcStateStatus, '9. ');
	ELSE
		sFrmWcStateStatus:= CONCAT( sFrmWcStateStatus, '');
	END_IF
	IF uiFrmWcState[iFrmNumber].9 THEN
		sFrmWcStateStatus:= CONCAT( sFrmWcStateStatus, '10. ');
	ELSE
		sFrmWcStateStatus:= CONCAT( sFrmWcStateStatus, '');
	END_IF
	IF uiFrmWcState[iFrmNumber].10 THEN
		sFrmWcStateStatus:= CONCAT( sFrmWcStateStatus, '11. ');
	ELSE
		sFrmWcStateStatus:= CONCAT( sFrmWcStateStatus, '');
	END_IF
	IF uiFrmWcState[iFrmNumber].11 THEN
		sFrmWcStateStatus:= CONCAT( sFrmWcStateStatus, '12. ');
	ELSE
		sFrmWcStateStatus:= CONCAT( sFrmWcStateStatus, '');
	END_IF
	IF uiFrmWcState[iFrmNumber].12 THEN
		sFrmWcStateStatus:= CONCAT( sFrmWcStateStatus, '13. ');
	ELSE
		sFrmWcStateStatus:= CONCAT( sFrmWcStateStatus, '');
	END_IF
	IF uiFrmWcState[iFrmNumber].13 THEN
		sFrmWcStateStatus:= CONCAT( sFrmWcStateStatus, '14. ');
	ELSE
		sFrmWcStateStatus:= CONCAT( sFrmWcStateStatus, '');
	END_IF
	IF uiFrmWcState[iFrmNumber].14 THEN
		sFrmWcStateStatus:= CONCAT( sFrmWcStateStatus, '15. ');
	ELSE
		sFrmWcStateStatus:= CONCAT( sFrmWcStateStatus, '');
	END_IF

	sFrmWcStateStatus:= CONCAT(sFrmWcStateStatus, 'EtherCAT command received. ' );

ELSIF uiFrmWcState[iFrmNumber]= 0 THEN
	sFrmWcStateStatus:= '';
END_IF

IF uiFrmWcState[iFrmNumber].15 THEN
	sFrmWcStateStatus:=  'Complete frame missing! ';
ELSE
	sFrmWcStateStatus:= CONCAT( sFrmWcStateStatus, '');
END_IF


IF sFrmWcStateStatus= '' THEN
	FrmWcState_Diagnosis:= TRUE;
ELSE
	FrmWcState_Diagnosis:= FALSE;
END_IF
END_METHOD

METHOD SlaveCount_Diagnosis : BOOL
VAR_INPUT
END_VAR
IF uiSlaveCount=uiCfgSlaveCount AND uiSlaveCount<>0 AND uiCfgSlaveCount<>0 THEN
	SlaveCount_Diagnosis:=TRUE;
ELSE
	SlaveCount_Diagnosis:=FALSE;
END_IF
END_METHOD

END_FUNCTION_BLOCK

// ---- POUs/ゴミ箱/P_Motion.TcPOU
PROGRAM P_Motion
VAR
	eAxis							:E_Axis;

END_VAR

	//---図形描画実行---
	IF GVL_MitsubishiCom.bToMcPowerOn=TRUE THEN;
		GVL_Motion.bWriteMoveStart:=GVL_MitsubishiCom.bFromWriteStart;
	END_IF

	//---ピック＆プレース実行---
	IF GVL_MitsubishiCom.bToMcPowerOn=TRUE THEN;
		GVL_Motion.bPickAndPlaceStart:=GVL_MitsubishiCom.bFromPickAndPlaceStart;
	END_IF
	
	//---アクションをコールして軸を起動---
	FOR eAxis:= E_Axis.X_Axis TO E_Axis.Gripper DO
		aMotion();
	END_FOR;

ACTION aMotion:
//パワーON
	GVL_Motion.fbMcPower[eAxis](
		Axis			:=GVL_Axis.stAxis[eAxis],
		Enable			:=GVL_Motion.bPower,
		Enable_Positive	:=GVL_Motion.bPower,
		Enable_Negative	:=GVL_Motion.bPower,
		Override		:=100,
		Status			=>,
		Busy			=>,
		Active			=>,
		Error			=>,
		ErrorID			=>
	);
	
//ホーミング
	GVL_Motion.fbMcMoveHome[eAxis](
		Axis			:=GVL_Axis.stAxis[eAxis],
		Execute			:=GVL_Motion.bHome,
		Position		:=0,
		Velocity		:=50,
		Done			=>,
		Busy			=>,
		Active			=>,
		CommandAborted	=>,
		Error			=>,
		ErrorID			=>
	);	

//定位置ジョグ
	GVL_Motion.fbMcMoveJog[eAxis](
		Axis			:=GVL_Axis.stAxis[eAxis],
		Execute			:=GVL_Motion.bJog[eAxis],
		Position		:=GVL_Motion.lrJogPosition[eAxis],
		Velocity		:=50,
		Done			=>,
		Busy			=>,
		Active			=>,
		CommandAborted	=>,
		Error			=>,
		ErrorID			=>
	);	

//連続ジョグ
	//起動
	GVL_Motion.fbMcMoveJogSub[eAxis](
		Axis			:=GVL_Axis.stAxis[eAxis],
	);
	//停止
	GVL_Motion.fbMCHaltJogSub[eAxis](
		Axis			:=GVL_Axis.stAxis[eAxis],
	);
	
//全軸一時停止
	GVL_Motion.fbMCHalt[eAxis](
		Axis			:=GVL_Axis.stAxis[eAxis],
		Execute			:=GVL_Motion.bHalt,
		Done			=>,
		Busy			=>,
		Active			=>,
		CommandAborted	=>,
		Error			=>,
		ErrorID			=>
	);

//全軸ストップ
	GVL_Motion.fbMCStop[eAxis](
		Axis			:=GVL_Axis.stAxis[eAxis],
		Execute			:=GVL_Motion.bStop,
		Done			=>,
		Busy			=>,
		Active			=>,
		CommandAborted	=>,
		Error			=>,
		ErrorID			=>
	);
	
//全軸リセット
	GVL_Motion.fbMcReset[eAxis](
		Axis			:=GVL_Axis.stAxis[eAxis],
		Execute			:=GVL_Motion.bReset,
		Done			=>,
		Busy			=>,
		Error			=>,
		ErrorID			=>
	);
END_ACTION

END_PROGRAM

// ---- POUs/ゴミ箱/P_PickAndPlace.TcPOU
PROGRAM P_PickAndPlace
VAR
	eStep				:E_PickAndPlaceStep:=E_PickAndPlaceStep.Stay;
	iStep				:INT:=0;
	fbMcMoveAbs			:ARRAY[E_Axis.X_Axis..E_Axis.Gripper] OF MC_MoveAbsolute;
	fbZAxisTargetPosCon	:FB_Z_Axis_TargetPositionConvert;
	
	XAxisTarget			:LREAL;
	YAxisTarget			:LREAL;
	ZAxisTarget			:LREAL:=270;
	GripperTarget		:LREAL:=70;
	
	ZAxisUpTarget		:LREAL:=200;
	ZAxisMidTarget		:LREAL:=235;
	
	AllAxisVelo			:LREAL;
	ZAxisTargetVelo		:LREAL;
	GripperVelo			:LREAL;
	
	i					:INT;
END_VAR

//Pick And Place Motin実行中か確認
IF eStep<>E_PickAndPlaceStep.Stay THEN
	
	//McMoveのコマンドアボートをチェック
	IF fbMcMoveAbs[E_Axis.X_Axis].CommandAborted=TRUE
		OR fbMcMoveAbs[E_Axis.Y_Axis].CommandAborted=TRUE
		OR fbMcMoveAbs[E_Axis.Z_Axis].CommandAborted=TRUE
		OR fbMcMoveAbs[E_Axis.Gripper].CommandAborted=TRUE THEN
			eStep:=E_PickAndPlaceStep.CommandAborted;
	END_IF
	
	//McMoveのエラーをチェック
	IF fbMcMoveAbs[E_Axis.X_Axis].Error=TRUE
		OR fbMcMoveAbs[E_Axis.Y_Axis].Error=TRUE
		OR fbMcMoveAbs[E_Axis.Z_Axis].Error=TRUE
		OR fbMcMoveAbs[E_Axis.Gripper].Error=TRUE THEN
			eStep:=E_PickAndPlaceStep.Error;
	END_IF

END_IF
	
CASE eStep OF

E_PickAndPlaceStep.Stay:(*初期値、bMoveがTrueになったらステップを進める*)

	IF GVL_Motion.bPickAndPlaceStart=TRUE THEN
		GVL_Motion.bAutoCameraTriger:=FALSE;
		GVL_Motion.bGetImageEnd:=FALSE;
		GVL_MitsubishiCom.bToPickAndPlaceMoving:=TRUE;
		eStep:=E_PickAndPlaceStep.GripperOpen;
	ELSE
		eStep:=E_PickAndPlaceStep.Stay;
	END_IF;

E_PickAndPlaceStep.GripperOpen:(*グリッパーを開ける*)
	
	fbMcMoveAbs[E_Axis.Gripper].Execute:=TRUE;
	fbMcMoveAbs[E_Axis.Gripper].Position:=0;
	fbMcMoveAbs[E_Axis.Gripper].Velocity:=7200;

	IF fbMcMoveAbs[E_Axis.Gripper].Done=TRUE THEN
		eStep:=E_PickAndPlaceStep.ZAxixZeroPos;
		fbMcMoveAbs[E_Axis.Gripper].Execute:=FALSE;
	END_IF;

E_PickAndPlaceStep.ZAxixZeroPos:(*Z軸をゼロポジションへ、衝突回避のためにまずZ軸を移動*)

	fbMcMoveAbs[E_Axis.Z_Axis].Execute:=TRUE;
	fbMcMoveAbs[E_Axis.Z_Axis].Position:=0;
	fbMcMoveAbs[E_Axis.Z_Axis].Velocity:=300;

	IF fbMcMoveAbs[E_Axis.Z_Axis].Done=TRUE THEN
		eStep:=E_PickAndPlaceStep.XYAxixShootingPos;
		fbMcMoveAbs[E_Axis.Z_Axis].Execute:=FALSE;
	END_IF;

E_PickAndPlaceStep.XYAxixShootingPos:(*Z軸移動後に、X,Y軸を撮影ポジションへ移動*)

	fbMcMoveAbs[E_Axis.X_Axis].Execute:=TRUE;
	fbMcMoveAbs[E_Axis.Y_Axis].Execute:=TRUE;
	fbMcMoveAbs[E_Axis.X_Axis].Position:=0;
	fbMcMoveAbs[E_Axis.Y_Axis].Position:=300;
	fbMcMoveAbs[E_Axis.X_Axis].Velocity:=300;
	fbMcMoveAbs[E_Axis.Y_Axis].Velocity:=300;
	
	IF fbMcMoveAbs[E_Axis.X_Axis].Done=TRUE AND fbMcMoveAbs[E_Axis.Y_Axis].Done=TRUE THEN
		eStep:=E_PickAndPlaceStep.Shooting;
		fbMcMoveAbs[E_Axis.X_Axis].Execute:=FALSE;
		fbMcMoveAbs[E_Axis.Y_Axis].Execute:=FALSE;
	END_IF;

E_PickAndPlaceStep.Shooting:(*カメラで画像を撮影*)
	
	GVL_Motion.bAutoCameraTriger:=TRUE;

	IF GVL_Motion.bGetImageEnd=TRUE THEN
		GVL_Motion.bAutoCameraTriger:=FALSE;
		GVL_Motion.bGetImageEnd:=FALSE;
		eStep:=E_PickAndPlaceStep.PickAndPlaceMotion_ResetVar;
	END_IF
	
E_PickAndPlaceStep.PickAndPlaceMotion_ResetVar:(*ピック＆プレース使用の変数をリセット*)
	
	//変数リセット
	i:=1;
	AllAxisVelo:=300;
	ZAxisTargetVelo:=50;
	GripperVelo:=3600;
	
	//ワークの数が0個ではないか確認
	IF ULINT_TO_INT(GVL_Vision.nDetectedNum) < i THEN
		eStep:=E_PickAndPlaceStep.ZAxixZeroPotision2;
	ELSE
		eStep:=E_PickAndPlaceStep.PickAndPlaceMotion_ValueCon;
	END_IF

E_PickAndPlaceStep.PickAndPlaceMotion_ValueCon:(*標値の変換実施*)
	//画像の座標をロボットの座標に変換X軸
	IF GVL_Vision.aMassCenter[i][0]<1052 THEN
		XAxisTarget:=0;
	ELSIF 4354<GVL_Vision.aMassCenter[i][0] THEN
		XAxisTarget:=300;
	ELSE
		XAxisTarget:=(300.0/(4354-1052))*(GVL_Vision.aMassCenter[i][0]-1052);
	END_IF

	//画像の座標をロボットの座標に変換Y軸
	IF GVL_Vision.aMassCenter[i][1]<146 THEN
		YAxisTarget:=0;
	ELSIF 3472<GVL_Vision.aMassCenter[i][1] THEN
		YAxisTarget:=300;
	ELSE
		YAxisTarget:=(300.0/(3472-146))*(GVL_Vision.aMassCenter[i][1]-146);
	END_IF
	
	//XY軸よりZ軸のターゲット座標値
	fbZAxisTargetPosCon(lrX_AxisTP		:=XAxisTarget,
						lrY_AxisTP		:=YAxisTarget,
						lrZ_AxisTP		:=ZAxisTarget,
						lrZ_AxisConTP	=>
						);

	eStep:=E_PickAndPlaceStep.PickAndPlaceMotion_XYAxisTargetPos;

	
E_PickAndPlaceStep.PickAndPlaceMotion_XYAxisTargetPos:(*XY軸をターゲットポジションへ*)
	fbMcMoveAbs[E_Axis.X_Axis].Execute:=TRUE;
	fbMcMoveAbs[E_Axis.Y_Axis].Execute:=TRUE;
	fbMcMoveAbs[E_Axis.X_Axis].Position:=XAxisTarget;
	fbMcMoveAbs[E_Axis.Y_Axis].Position:=YAxisTarget;
	fbMcMoveAbs[E_Axis.X_Axis].Velocity:=AllAxisVelo;
	fbMcMoveAbs[E_Axis.Y_Axis].Velocity:=AllAxisVelo;
	
	IF fbMcMoveAbs[E_Axis.X_Axis].Done=TRUE AND fbMcMoveAbs[E_Axis.Y_Axis].Done=TRUE THEN
		eStep:=E_PickAndPlaceStep.PickAndPlaceMotion_ZAxisUpPos;
		fbMcMoveAbs[E_Axis.X_Axis].Execute:=FALSE;
		fbMcMoveAbs[E_Axis.Y_Axis].Execute:=FALSE;
	END_IF;

		
E_PickAndPlaceStep.PickAndPlaceMotion_ZAxisUpPos:(*Z軸を上昇位置へ*)

	fbMcMoveAbs[E_Axis.Z_Axis].Execute:=TRUE;
	fbMcMoveAbs[E_Axis.Z_Axis].Position:=ZAxisUpTarget;
	fbMcMoveAbs[E_Axis.Z_Axis].Velocity:=AllAxisVelo;

	IF fbMcMoveAbs[E_Axis.Z_Axis].Done=TRUE THEN
		eStep:=E_PickAndPlaceStep.PickAndPlaceMotion_ZAxisTargetPos;
		fbMcMoveAbs[E_Axis.Z_Axis].Execute:=FALSE;
	END_IF;

	
E_PickAndPlaceStep.PickAndPlaceMotion_ZAxisTargetPos:(*Z軸をターゲットポジションへ*)

	CASE iStep OF
	
	0:
		fbMcMoveAbs[E_Axis.Z_Axis].Execute:=TRUE;
		fbMcMoveAbs[E_Axis.Z_Axis].Position:=fbZAxisTargetPosCon.lrZ_AxisConTP-10;
		fbMcMoveAbs[E_Axis.Z_Axis].Velocity:=AllAxisVelo;
	
		IF fbMcMoveAbs[E_Axis.Z_Axis].Done=TRUE THEN
			iStep:=1;
			fbMcMoveAbs[E_Axis.Z_Axis].Execute:=FALSE;
		END_IF;
	
	1:
		fbMcMoveAbs[E_Axis.Z_Axis].Execute:=TRUE;
		fbMcMoveAbs[E_Axis.Z_Axis].Position:=fbZAxisTargetPosCon.lrZ_AxisConTP;
		fbMcMoveAbs[E_Axis.Z_Axis].Velocity:=ZAxisTargetVelo;
	
		IF fbMcMoveAbs[E_Axis.Z_Axis].Done=TRUE THEN
			eStep:=E_PickAndPlaceStep.PickAndPlaceMotion_GripperGrip;
			iStep:=0;
			fbMcMoveAbs[E_Axis.Z_Axis].Execute:=FALSE;
		END_IF;
	
	END_CASE

	
E_PickAndPlaceStep.PickAndPlaceMotion_GripperGrip:(*グリッパーを閉じてマグネットを掴む*)
	fbMcMoveAbs[E_Axis.Gripper].Execute:=TRUE;
	fbMcMoveAbs[E_Axis.Gripper].Position:=GripperTarget;
	fbMcMoveAbs[E_Axis.Gripper].Velocity:=GripperVelo;

	IF fbMcMoveAbs[E_Axis.Gripper].Done=TRUE THEN
		eStep:=E_PickAndPlaceStep.PickAndPlaceMotion_ZAxisUpPos2;
		fbMcMoveAbs[E_Axis.Gripper].Execute:=FALSE;
	END_IF;
		
		
E_PickAndPlaceStep.PickAndPlaceMotion_ZAxisUpPos2:(*Z軸を上昇位置へ*)

	fbMcMoveAbs[E_Axis.Z_Axis].Execute:=TRUE;
	fbMcMoveAbs[E_Axis.Z_Axis].Position:=ZAxisUpTarget;
	fbMcMoveAbs[E_Axis.Z_Axis].Velocity:=AllAxisVelo;

	IF fbMcMoveAbs[E_Axis.Z_Axis].Done=TRUE THEN
		eStep:=E_PickAndPlaceStep.PickAndPlaceMotion_XYAxis300Pos;
		fbMcMoveAbs[E_Axis.Z_Axis].Execute:=FALSE;
	END_IF;
		
	
E_PickAndPlaceStep.PickAndPlaceMotion_XYAxis300Pos:(*XY軸を300ポジションへ、300にはお皿がおいてあるはず*)
	fbMcMoveAbs[E_Axis.X_Axis].Execute:=TRUE;
	fbMcMoveAbs[E_Axis.Y_Axis].Execute:=TRUE;
	fbMcMoveAbs[E_Axis.X_Axis].Position:=300;
	fbMcMoveAbs[E_Axis.Y_Axis].Position:=300;
	fbMcMoveAbs[E_Axis.X_Axis].Velocity:=AllAxisVelo;
	fbMcMoveAbs[E_Axis.Y_Axis].Velocity:=AllAxisVelo;
	
	IF fbMcMoveAbs[E_Axis.X_Axis].Done=TRUE AND fbMcMoveAbs[E_Axis.Y_Axis].Done=TRUE THEN
		eStep:=E_PickAndPlaceStep.PickAndPlaceMotion_ZAxisMidPos;
		fbMcMoveAbs[E_Axis.X_Axis].Execute:=FALSE;
		fbMcMoveAbs[E_Axis.Y_Axis].Execute:=FALSE;
	END_IF;


E_PickAndPlaceStep.PickAndPlaceMotion_ZAxisMidPos:(*Z軸をマグネットをリリースする高さへ*)

	fbMcMoveAbs[E_Axis.Z_Axis].Execute:=TRUE;
	fbMcMoveAbs[E_Axis.Z_Axis].Position:=ZAxisMidTarget;
	fbMcMoveAbs[E_Axis.Z_Axis].Velocity:=AllAxisVelo;

	IF fbMcMoveAbs[E_Axis.Z_Axis].Done=TRUE THEN
		eStep:=E_PickAndPlaceStep.PickAndPlaceMotion_GripperOpen;
		fbMcMoveAbs[E_Axis.Z_Axis].Execute:=FALSE;
	END_IF;


E_PickAndPlaceStep.PickAndPlaceMotion_GripperOpen:(*グリッパーを開けてマグネットをお皿へ*)
	
	fbMcMoveAbs[E_Axis.Gripper].Execute:=TRUE;
	fbMcMoveAbs[E_Axis.Gripper].Position:=0;
	fbMcMoveAbs[E_Axis.Gripper].Velocity:=GripperVelo;

	IF fbMcMoveAbs[E_Axis.Gripper].Done=TRUE THEN
		eStep:=E_PickAndPlaceStep.PickAndPlaceMotion_ZAxisUpPos3;
		fbMcMoveAbs[E_Axis.Gripper].Execute:=FALSE;
	END_IF;


E_PickAndPlaceStep.PickAndPlaceMotion_ZAxisUpPos3:(*Z軸を上昇位置へ*)

	fbMcMoveAbs[E_Axis.Z_Axis].Execute:=TRUE;
	fbMcMoveAbs[E_Axis.Z_Axis].Position:=ZAxisUpTarget;
	fbMcMoveAbs[E_Axis.Z_Axis].Velocity:=AllAxisVelo;

	IF fbMcMoveAbs[E_Axis.Z_Axis].Done=TRUE THEN
		eStep:=E_PickAndPlaceStep.PickAndPlaceMotion_NextCheck;
		fbMcMoveAbs[E_Axis.Z_Axis].Execute:=FALSE;
	END_IF;
	
	
E_PickAndPlaceStep.PickAndPlaceMotion_NextCheck:(*次のマグネットがあるか確認、無ければ終わり、あればピック＆プレースの最初へ戻る*)

	i:=i+1;
	
	IF ULINT_TO_INT(GVL_Vision.nDetectedNum) < i THEN
		eStep:=E_PickAndPlaceStep.ZAxixZeroPotision2;
	ELSE
		eStep:=E_PickAndPlaceStep.PickAndPlaceMotion_ValueCon;
	END_IF


E_PickAndPlaceStep.ZAxixZeroPotision2:(*Z軸をゼロポジションへ、衝突回避のためにまずZ軸を移動*)

	fbMcMoveAbs[E_Axis.Z_Axis].Execute:=TRUE;
	fbMcMoveAbs[E_Axis.Z_Axis].Position:=0;
	fbMcMoveAbs[E_Axis.Z_Axis].Velocity:=300;

	IF fbMcMoveAbs[E_Axis.Z_Axis].Done=TRUE THEN
		eStep:=E_PickAndPlaceStep.XYAxixZeroPotision2;
		fbMcMoveAbs[E_Axis.Z_Axis].Execute:=FALSE;
	END_IF;
	
E_PickAndPlaceStep.XYAxixZeroPotision2:(*Z軸移動後に、X,Y軸をゼロポジションへ移動*)

	fbMcMoveAbs[E_Axis.X_Axis].Execute:=TRUE;
	fbMcMoveAbs[E_Axis.Y_Axis].Execute:=TRUE;
	fbMcMoveAbs[E_Axis.X_Axis].Position:=0;
	fbMcMoveAbs[E_Axis.Y_Axis].Position:=0;
	fbMcMoveAbs[E_Axis.X_Axis].Velocity:=300;
	fbMcMoveAbs[E_Axis.Y_Axis].Velocity:=300;
	
	IF fbMcMoveAbs[E_Axis.X_Axis].Done=TRUE AND fbMcMoveAbs[E_Axis.Y_Axis].Done=TRUE THEN
		eStep:=E_PickAndPlaceStep.Stay;
		GVL_MitsubishiCom.bToPickAndPlaceMoving:=FALSE;
		fbMcMoveAbs[E_Axis.X_Axis].Execute:=FALSE;
		fbMcMoveAbs[E_Axis.Y_Axis].Execute:=FALSE;
	END_IF;
	
E_PickAndPlaceStep.CommandAborted://McMoveコマンドアボート時の処理	

	iStep:=0;
	fbMcMoveAbs[E_Axis.X_Axis].Execute:=FALSE;
	fbMcMoveAbs[E_Axis.Y_Axis].Execute:=FALSE;
	fbMcMoveAbs[E_Axis.Z_Axis].Execute:=FALSE;
	fbMcMoveAbs[E_Axis.Gripper].Execute:=FALSE;
	
	GVL_MitsubishiCom.bToAutoMoveResetting:=FALSE;

	IF fbMcMoveAbs[E_Axis.X_Axis].CommandAborted=FALSE
		AND fbMcMoveAbs[E_Axis.Y_Axis].CommandAborted=FALSE
		AND fbMcMoveAbs[E_Axis.Z_Axis].CommandAborted=FALSE
		AND fbMcMoveAbs[E_Axis.Gripper].CommandAborted=FALSE THEN
			eStep:=E_PickAndPlaceStep.Reset;
	END_IF

E_PickAndPlaceStep.Error://McMoveエラー時の処理	

	iStep:=0;
	fbMcMoveAbs[E_Axis.X_Axis].Execute:=FALSE;
	fbMcMoveAbs[E_Axis.Y_Axis].Execute:=FALSE;
	fbMcMoveAbs[E_Axis.Z_Axis].Execute:=FALSE;
	fbMcMoveAbs[E_Axis.Gripper].Execute:=FALSE;
	
	GVL_MitsubishiCom.bToAutoMoveResetting:=FALSE;

	if fbMcMoveAbs[E_Axis.X_Axis].Error=FALSE
		AND fbMcMoveAbs[E_Axis.Y_Axis].Error=FALSE
		AND fbMcMoveAbs[E_Axis.Z_Axis].Error=FALSE
		AND fbMcMoveAbs[E_Axis.Gripper].Error=FALSE THEN
			eStep:=E_PickAndPlaceStep.Reset;
	END_IF	
	
E_PickAndPlaceStep.Reset://McMoveのコマンドアボートorエラー後のリセット動作

	CASE iStep OF

	0:
		IF GVL_MitsubishiCom.bFromAutoMoveReset=TRUE AND MAIN.fb3AxisRobot.fbMachineState.bStopMachine=FALSE THEN
			GVL_MitsubishiCom.bToAutoMoveResetting:=TRUE;
			iStep:=1;
		END_IF

	1:
		fbMcMoveAbs[E_Axis.Gripper].Execute:=TRUE;
		fbMcMoveAbs[E_Axis.Gripper].Position:=0;
		fbMcMoveAbs[E_Axis.Gripper].Velocity:=150;

		IF fbMcMoveAbs[E_Axis.Gripper].Done=TRUE THEN
			iStep:=2;
			fbMcMoveAbs[E_Axis.Gripper].Execute:=FALSE;
		END_IF;

	2:
		fbMcMoveAbs[E_Axis.Z_Axis].Execute:=TRUE;
		fbMcMoveAbs[E_Axis.Z_Axis].Position:=0;
		fbMcMoveAbs[E_Axis.Z_Axis].Velocity:=150;

		IF fbMcMoveAbs[E_Axis.Z_Axis].Done=TRUE THEN
			iStep:=3;
			fbMcMoveAbs[E_Axis.Z_Axis].Execute:=FALSE;
		END_IF;

	3:
		fbMcMoveAbs[E_Axis.X_Axis].Execute:=TRUE;
		fbMcMoveAbs[E_Axis.Y_Axis].Execute:=TRUE;
		fbMcMoveAbs[E_Axis.X_Axis].Position:=0;
		fbMcMoveAbs[E_Axis.Y_Axis].Position:=0;
		fbMcMoveAbs[E_Axis.X_Axis].Velocity:=150;
		fbMcMoveAbs[E_Axis.Y_Axis].Velocity:=150;

		IF fbMcMoveAbs[E_Axis.X_Axis].Done=TRUE AND fbMcMoveAbs[E_Axis.Y_Axis].Done=TRUE THEN
			fbMcMoveAbs[E_Axis.X_Axis].Execute:=FALSE;
			fbMcMoveAbs[E_Axis.Y_Axis].Execute:=FALSE;
			iStep:=0;
			eStep:=E_PickAndPlaceStep.Stay;

			GVL_MitsubishiCom.bToPickAndPlaceMoving:=FALSE;
			GVL_MitsubishiCom.bToAutoMoveResetting:=FALSE;
		END_IF;

	END_CASE
	
END_CASE;

	aMotion();

ACTION aMotion:
//各軸とグリッパーの駆動用
	//メイン
	fbMcMoveAbs[E_Axis.X_Axis](
		Axis			:=GVL_Axis.stAxis[E_Axis.X_Axis],
		BufferMode		:=MC_BlendingNext,
	);

	fbMcMoveAbs[E_Axis.Y_Axis](
		Axis			:=GVL_Axis.stAxis[E_Axis.Y_Axis],
		BufferMode		:=MC_BlendingNext,
	);

	fbMcMoveAbs[E_Axis.Z_Axis](
		Axis			:=GVL_Axis.stAxis[E_Axis.Z_Axis],
		BufferMode		:=MC_BlendingNext,
	);
	
	fbMcMoveAbs[E_Axis.Gripper](
		Axis			:=GVL_Axis.stAxis[E_Axis.Gripper],
		BufferMode		:=MC_BlendingNext,
	);
END_ACTION

END_PROGRAM
